C05467=1086.034,-74.611,447.064,174.286,17.662,152.886
C05468=1086.028,-74.861,447.075,174.284,17.661,152.887
C05469=1086.021,-75.111,447.086,174.282,17.660,152.887
C05470=1086.016,-75.360,447.097,174.281,17.658,152.887
C05471=1086.010,-75.610,447.108,174.279,17.657,152.887
C05472=1086.004,-75.860,447.119,174.278,17.656,152.887
C05473=1085.998,-76.110,447.130,174.277,17.655,152.887
C05474=1085.992,-76.359,447.141,174.275,17.654,152.887
C05475=1085.986,-76.608,447.151,174.274,17.653,152.887
C05476=1085.979,-76.858,447.162,174.272,17.652,152.887
C05477=1085.974,-77.108,447.173,174.271,17.650,152.887
C05478=1085.968,-77.358,447.183,174.269,17.649,152.887
C05479=1085.962,-77.607,447.194,174.268,17.648,152.887
C05480=1085.956,-77.858,447.205,174.266,17.646,152.887
C05481=1085.950,-78.107,447.215,174.265,17.645,152.887
C05482=1085.944,-78.356,447.226,174.263,17.644,152.887
C05483=1085.938,-78.607,447.238,174.261,17.643,152.887
C05484=1085.932,-78.856,447.248,174.260,17.642,152.887
C05485=1085.926,-79.105,447.259,174.258,17.640,152.887
C05486=1085.921,-79.356,447.270,174.257,17.639,152.887
C05487=1085.914,-79.605,447.280,174.255,17.638,152.888
C05488=1085.908,-79.855,447.291,174.254,17.636,152.888
C05489=1085.902,-80.104,447.302,174.252,17.635,152.888
C05490=1085.896,-80.354,447.313,174.250,17.634,152.888
C05491=1085.889,-80.604,447.323,174.250,17.634,152.888
C05492=1085.883,-80.879,447.335,174.247,17.631,152.888
C05493=1085.876,-81.154,447.346,174.246,17.630,152.888
C05494=1085.870,-81.429,447.358,174.244,17.629,152.888
C05495=1085.863,-81.705,447.371,174.243,17.628,152.888
C05496=1085.857,-81.955,447.381,174.241,17.627,152.888
C05497=1085.851,-82.204,447.391,174.239,17.626,152.888
C05498=1085.845,-82.454,447.402,174.238,17.625,152.888
C05499=1085.839,-82.704,447.413,174.236,17.623,152.888
C05500=1085.832,-82.953,447.423,174.235,17.622,152.888
C05501=1085.827,-83.203,447.434,174.233,17.621,152.889
C05502=1085.820,-83.452,447.444,174.232,17.620,152.889
C05503=1085.814,-83.703,447.455,174.231,17.619,152.889
C05504=1085.808,-83.952,447.466,174.229,17.618,152.889
C05505=1085.802,-84.202,447.476,174.227,17.617,152.889
C05506=1085.796,-84.451,447.486,174.226,17.616,152.889
C05507=1085.790,-84.702,447.498,174.224,17.615,152.889
C05508=1085.784,-84.951,447.507,174.223,17.613,152.889
C05509=1085.778,-85.201,447.518,174.221,17.612,152.889
C05510=1085.771,-85.450,447.528,174.219,17.611,152.889
C05511=1085.766,-85.699,447.539,174.218,17.610,152.889
C05512=1085.760,-85.950,447.550,174.216,17.608,152.889
C05513=1085.753,-86.199,447.560,174.216,17.608,152.889
C05514=1085.747,-86.449,447.571,174.214,17.607,152.889
C05515=1085.741,-86.699,447.581,174.212,17.606,152.890
C05516=1085.736,-86.948,447.591,174.211,17.604,152.890
C05517=1085.729,-87.198,447.603,174.209,17.603,152.890
C05518=1085.723,-87.448,447.612,174.208,17.602,152.890
C05519=1085.717,-87.698,447.623,174.206,17.601,152.890
C05520=1085.711,-87.947,447.633,174.204,17.600,152.890
C05521=1085.705,-88.197,447.644,174.203,17.599,152.890
C05522=1085.699,-88.446,447.654,174.201,17.597,152.890
C05523=1085.693,-88.697,447.664,174.200,17.596,152.890
C05524=1085.687,-88.947,447.675,174.199,17.595,152.890
C05525=1085.681,-89.196,447.686,174.197,17.594,152.890
C05526=1085.675,-89.446,447.696,174.195,17.593,152.890
C05527=1085.669,-89.695,447.706,174.194,17.592,152.891
C05528=1085.663,-89.945,447.716,174.192,17.591,152.891
C05529=1085.656,-90.195,447.727,174.191,17.590,152.891
C05530=1085.650,-90.444,447.738,174.189,17.589,152.891
C05531=1085.645,-90.695,447.748,174.187,17.587,152.891
C05532=1085.639,-90.944,447.758,174.187,17.587,152.891
C05533=1085.633,-91.194,447.768,174.185,17.586,152.891
C05534=1085.627,-91.443,447.779,174.183,17.585,152.891
C05535=1085.621,-91.693,447.789,174.182,17.583,152.891
C05536=1085.615,-91.942,447.799,174.180,17.582,152.891
C05537=1085.609,-92.193,447.810,174.179,17.581,152.891
C05538=1085.602,-92.442,447.820,174.177,17.580,152.891
C05539=1085.597,-92.692,447.830,174.175,17.579,152.892
C05540=1085.590,-92.942,447.840,174.174,17.578,152.892
C05541=1085.585,-93.192,447.850,174.173,17.577,152.892
C05542=1085.578,-93.441,447.861,174.171,17.576,152.892
C05543=1085.573,-93.691,447.871,174.170,17.575,152.892
C05544=1085.567,-93.940,447.881,174.168,17.574,152.892
C05545=1085.561,-94.190,447.891,174.166,17.573,152.892
C05546=1085.555,-94.439,447.902,174.165,17.572,152.892
C05547=1085.549,-94.690,447.912,174.163,17.570,152.892
C05548=1085.543,-94.939,447.922,174.162,17.570,152.892
C05549=1085.537,-95.189,447.932,174.161,17.569,152.892
C05550=1085.530,-95.439,447.943,174.159,17.568,152.893
C05551=1085.525,-95.689,447.953,174.157,17.567,152.893
C05552=1085.518,-95.938,447.963,174.156,17.566,152.893
C05553=1085.513,-96.188,447.973,174.154,17.564,152.893
C05554=1085.507,-96.438,447.983,174.153,17.563,152.893
C05555=1085.501,-96.687,447.994,174.152,17.563,152.893
C05556=1085.494,-96.964,448.005,174.150,17.561,152.893
C05557=1085.488,-97.242,448.016,174.148,17.560,152.893
C05558=1085.481,-97.520,448.028,174.146,17.559,152.893
C05559=1085.474,-97.797,448.038,174.144,17.558,152.893
C05560=1085.469,-98.047,448.049,174.144,17.557,152.894
C05561=1085.462,-98.297,448.059,174.142,17.556,152.894
C05562=1085.455,-98.547,448.069,174.140,17.555,152.894
C05563=1085.450,-98.797,448.079,174.139,17.554,152.894
C05564=1085.444,-99.046,448.089,174.137,17.553,152.894
C05565=1085.437,-99.296,448.099,174.135,17.552,152.894
C05566=1085.432,-99.546,448.109,174.134,17.551,152.894
C05567=1085.425,-99.795,448.119,174.133,17.550,152.894
C05568=1085.419,-100.045,448.129,174.131,17.549,152.894
C05569=1085.414,-100.295,448.139,174.129,17.548,152.894
C05570=1085.407,-100.544,448.149,174.128,17.547,152.895
C05571=1085.401,-100.794,448.159,174.126,17.546,152.895
C05572=1085.395,-101.044,448.168,174.125,17.546,152.895
C05573=1085.389,-101.293,448.179,174.123,17.545,152.895
C05574=1085.383,-101.543,448.189,174.122,17.544,152.895
C05575=1085.377,-101.793,448.198,174.120,17.543,152.895
C05576=1085.371,-102.043,448.208,174.118,17.542,152.895
C05577=1085.365,-102.292,448.219,174.117,17.541,152.895
C05578=1085.359,-102.542,448.228,174.116,17.540,152.896
C05579=1085.353,-102.792,448.238,174.114,17.539,152.896
C05580=1085.347,-103.041,448.249,174.113,17.538,152.896
C05581=1085.341,-103.291,448.258,174.111,17.537,152.896
C05582=1085.335,-103.541,448.268,174.109,17.536,152.896
C05583=1085.328,-103.791,448.278,174.108,17.535,152.896
C05584=1085.323,-104.041,448.288,174.107,17.535,152.896
C05585=1085.317,-104.290,448.298,174.105,17.534,152.896
C05586=1085.310,-104.540,448.308,174.103,17.533,152.897
C05587=1085.304,-104.789,448.317,174.102,17.532,152.897
C05588=1085.298,-105.039,448.327,174.100,17.531,152.897
C05589=1085.292,-105.289,448.338,174.099,17.530,152.897
C05590=1085.286,-105.538,448.347,174.097,17.529,152.897
C05591=1085.280,-105.788,448.357,174.096,17.528,152.897
C05592=1085.274,-106.038,448.366,174.094,17.527,152.897
C05593=1085.268,-106.288,448.376,174.092,17.526,152.897
C05594=1085.262,-106.537,448.387,174.091,17.526,152.898
C05595=1085.256,-106.787,448.396,174.090,17.525,152.898
C05596=1085.250,-107.037,448.406,174.088,17.524,152.898
C05597=1085.243,-107.287,448.415,174.086,17.523,152.898
C05598=1085.237,-107.537,448.425,174.084,17.522,152.898
C05599=1085.232,-107.787,448.435,174.084,17.522,152.898
C05600=1085.226,-108.036,448.445,174.082,17.521,152.898
C05601=1085.219,-108.286,448.455,174.080,17.519,152.898
C05602=1085.213,-108.535,448.465,174.079,17.518,152.899
C05603=1085.207,-108.785,448.474,174.078,17.518,152.899
C05604=1085.201,-109.035,448.484,174.076,17.517,152.899
C05605=1085.194,-109.285,448.493,174.074,17.516,152.899
C05606=1085.188,-109.535,448.503,174.073,17.515,152.899
C05607=1085.182,-109.784,448.512,174.071,17.515,152.899
C05608=1085.176,-110.034,448.522,174.070,17.514,152.899
C05609=1085.169,-110.283,448.532,174.068,17.513,152.900
C05610=1085.164,-110.534,448.542,174.067,17.512,152.900
C05611=1085.158,-110.783,448.552,174.065,17.511,152.900
C05612=1085.152,-111.033,448.562,174.064,17.511,152.900
C05613=1085.145,-111.283,448.571,174.062,17.510,152.900
C05614=1085.139,-111.533,448.581,174.060,17.509,152.900
C05615=1085.133,-111.783,448.590,174.059,17.508,152.900
C05616=1085.128,-112.032,448.600,174.057,17.507,152.901
C05617=1085.121,-112.281,448.609,174.056,17.507,152.901
C05618=1085.115,-112.531,448.619,174.054,17.506,152.901
C05619=1085.109,-112.781,448.628,174.052,17.505,152.901
C05620=1085.103,-113.054,448.639,174.051,17.504,152.901
C05621=1085.095,-113.327,448.650,174.049,17.503,152.901
C05622=1085.089,-113.600,448.660,174.047,17.502,152.902
C05623=1085.082,-113.873,448.670,174.046,17.501,152.902
C05624=1085.076,-114.123,448.680,174.045,17.501,152.902
C05625=1085.070,-114.373,448.689,174.043,17.500,152.902
C05626=1085.064,-114.622,448.699,174.041,17.499,152.902
C05627=1085.058,-114.872,448.708,174.040,17.498,152.902
C05628=1085.052,-115.122,448.718,174.038,17.498,152.902
C05629=1085.046,-115.371,448.727,174.037,17.497,152.903
C05630=1085.040,-115.621,448.737,174.035,17.497,152.903
C05631=1085.033,-115.871,448.746,174.033,17.495,152.903
C05632=1085.027,-116.121,448.756,174.032,17.495,152.903
C05633=1085.021,-116.371,448.766,174.030,17.494,152.903
C05634=1085.015,-116.620,448.775,174.029,17.493,152.903
C05635=1085.009,-116.870,448.785,174.027,17.492,152.903
C05636=1085.003,-117.120,448.793,174.026,17.492,152.904
C05637=1084.997,-117.370,448.803,174.024,17.491,152.904
C05638=1084.990,-117.619,448.812,174.022,17.491,152.904
C05639=1084.984,-117.869,448.821,174.022,17.490,152.904
C05640=1084.978,-118.119,448.831,174.020,17.489,152.904
C05641=1084.972,-118.369,448.840,174.018,17.489,152.905
C05642=1084.966,-118.618,448.850,174.016,17.487,152.905
C05643=1084.959,-118.868,448.860,174.015,17.487,152.905
C05644=1084.954,-119.117,448.869,174.014,17.486,152.905
C05645=1084.948,-119.367,448.878,174.012,17.486,152.905
C05646=1084.942,-119.617,448.887,174.010,17.485,152.905
C05647=1084.936,-119.867,448.897,174.009,17.484,152.905
C05648=1084.929,-120.117,448.906,174.007,17.484,152.906
C05649=1084.923,-120.367,448.915,174.006,17.483,152.906
C05650=1084.916,-120.616,448.925,174.004,17.483,152.906
C05651=1084.911,-120.865,448.934,174.003,17.482,152.906
C05652=1084.905,-121.116,448.943,174.001,17.481,152.906
C05653=1084.899,-121.366,448.952,173.999,17.480,152.906
C05654=1084.893,-121.615,448.962,173.998,17.480,152.907
C05655=1084.886,-121.865,448.971,173.996,17.479,152.907
C05656=1084.880,-122.115,448.981,173.995,17.478,152.907
C05657=1084.874,-122.364,448.990,173.994,17.478,152.907
C05658=1084.868,-122.614,448.999,173.992,17.477,152.907
C05659=1084.862,-122.864,449.008,173.990,17.476,152.908
C05660=1084.856,-123.114,449.018,173.988,17.476,152.908
C05661=1084.849,-123.363,449.027,173.987,17.475,152.908
C05662=1084.843,-123.614,449.036,173.985,17.475,152.908
C05663=1084.837,-123.863,449.045,173.984,17.474,152.908
C05664=1084.831,-124.113,449.054,173.983,17.474,152.908
C05665=1084.825,-124.362,449.064,173.981,17.472,152.909
C05666=1084.819,-124.613,449.073,173.979,17.472,152.909
C05667=1084.812,-124.862,449.082,173.978,17.471,152.909
C05668=1084.807,-125.111,449.091,173.976,17.471,152.909
C05669=1084.801,-125.361,449.101,173.975,17.470,152.909
C05670=1084.794,-125.611,449.109,173.973,17.469,152.910
C05671=1084.788,-125.861,449.118,173.972,17.469,152.910
C05672=1084.782,-126.111,449.128,173.970,17.468,152.910
C05673=1084.775,-126.361,449.137,173.968,17.468,152.910
C05674=1084.769,-126.610,449.145,173.967,17.467,152.910
C05675=1084.763,-126.860,449.155,173.965,17.467,152.910
C05676=1084.757,-127.110,449.165,173.963,17.466,152.911
C05677=1084.750,-127.360,449.173,173.963,17.466,152.911
C05678=1084.744,-127.610,449.182,173.961,17.465,152.911
C05679=1084.739,-127.859,449.192,173.959,17.464,152.911
C05680=1084.733,-128.116,449.201,173.958,17.464,152.911
C05681=1084.731,-128.373,449.211,173.957,17.462,152.911
C05682=1084.733,-128.628,449.224,173.956,17.459,152.911
C05683=1084.740,-128.881,449.237,173.955,17.454,152.910
C05684=1084.338,-128.903,449.105,173.912,17.569,152.940
C05685=1084.332,-128.650,449.091,173.912,17.573,152.941
C05686=1084.328,-128.394,449.079,173.912,17.577,152.941
C05687=1084.331,-128.138,449.068,173.914,17.578,152.941
C05688=1084.335,-127.881,449.059,173.915,17.579,152.941
C05689=1084.342,-127.632,449.050,173.917,17.580,152.941
C05690=1084.348,-127.382,449.040,173.918,17.580,152.941
C05691=1084.354,-127.132,449.031,173.920,17.581,152.941
C05692=1084.361,-126.882,449.022,173.922,17.582,152.941
C05693=1084.367,-126.633,449.013,173.923,17.582,152.940
C05694=1084.373,-126.383,449.004,173.925,17.583,152.940
C05695=1084.379,-126.133,448.995,173.927,17.584,152.940
C05696=1084.386,-125.883,448.986,173.928,17.584,152.940
C05697=1084.392,-125.633,448.977,173.929,17.585,152.940
C05698=1084.397,-125.384,448.968,173.931,17.585,152.939
C05699=1084.404,-125.134,448.959,173.933,17.586,152.939
C05700=1084.410,-124.884,448.949,173.934,17.586,152.939
C05701=1084.416,-124.634,448.940,173.936,17.587,152.939
C05702=1084.422,-124.384,448.931,173.938,17.588,152.939
C05703=1084.428,-124.135,448.922,173.938,17.588,152.939
C05704=1084.435,-123.886,448.913,173.940,17.589,152.938
C05705=1084.441,-123.635,448.904,173.942,17.590,152.938
C05706=1084.447,-123.385,448.894,173.944,17.590,152.938
C05707=1084.453,-123.136,448.885,173.945,17.591,152.938
C05708=1084.459,-122.886,448.875,173.947,17.592,152.938
C05709=1084.466,-122.637,448.867,173.948,17.593,152.937
C05710=1084.471,-122.387,448.858,173.949,17.593,152.937
C05711=1084.478,-122.137,448.848,173.951,17.594,152.937
C05712=1084.484,-121.887,448.839,173.953,17.594,152.937
C05713=1084.490,-121.637,448.829,173.955,17.595,152.937
C05714=1084.496,-121.387,448.819,173.956,17.595,152.937
C05715=1084.501,-121.138,448.811,173.957,17.596,152.936
C05716=1084.508,-120.888,448.802,173.959,17.597,152.936
C05717=1084.514,-120.638,448.792,173.961,17.598,152.936
C05718=1084.521,-120.389,448.783,173.962,17.598,152.936
C05719=1084.527,-120.139,448.773,173.964,17.599,152.936
C05720=1084.533,-119.889,448.764,173.965,17.600,152.936
C05721=1084.538,-119.639,448.755,173.966,17.601,152.936
C05722=1084.544,-119.390,448.746,173.968,17.601,152.935
C05723=1084.551,-119.140,448.736,173.970,17.602,152.935
C05724=1084.557,-118.890,448.727,173.972,17.603,152.935
C05725=1084.564,-118.640,448.718,173.973,17.603,152.935
C05726=1084.570,-118.391,448.708,173.975,17.604,152.935
C05727=1084.576,-118.141,448.698,173.976,17.605,152.934
C05728=1084.582,-117.891,448.689,173.978,17.606,152.934
C05729=1084.588,-117.642,448.680,173.979,17.606,152.934
C05730=1084.594,-117.392,448.671,173.981,17.607,152.934
C05731=1084.600,-117.142,448.661,173.982,17.608,152.934
C05732=1084.606,-116.892,448.652,173.984,17.608,152.934
C05733=1084.612,-116.642,448.642,173.985,17.609,152.934
C05734=1084.618,-116.392,448.632,173.987,17.610,152.933
C05735=1084.624,-116.143,448.623,173.989,17.611,152.933
C05736=1084.631,-115.893,448.613,173.990,17.612,152.933
C05737=1084.638,-115.643,448.604,173.991,17.612,152.933
C05738=1084.643,-115.394,448.595,173.993,17.613,152.933
C05739=1084.649,-115.144,448.586,173.995,17.614,152.933
C05740=1084.655,-114.895,448.576,173.996,17.615,152.932
C05741=1084.662,-114.645,448.566,173.998,17.615,152.932
C05742=1084.668,-114.395,448.557,173.999,17.616,152.932
C05743=1084.674,-114.145,448.547,174.001,17.617,152.932
C05744=1084.680,-113.895,448.538,174.003,17.617,152.932
C05745=1084.686,-113.622,448.527,174.004,17.619,152.932
C05746=1084.693,-113.348,448.516,174.005,17.619,152.932
C05747=1084.700,-113.075,448.506,174.007,17.620,152.931
C05748=1084.706,-112.802,448.496,174.009,17.621,152.931
C05749=1084.712,-112.552,448.486,174.011,17.622,152.931
C05750=1084.718,-112.303,448.477,174.012,17.623,152.931
C05751=1084.725,-112.053,448.467,174.014,17.624,152.931
C05752=1084.731,-111.803,448.458,174.015,17.624,152.931
C05753=1084.737,-111.553,448.448,174.017,17.625,152.931
C05754=1084.743,-111.303,448.438,174.018,17.626,152.930
C05755=1084.749,-111.054,448.429,174.020,17.627,152.930
C05756=1084.755,-110.804,448.419,174.022,17.628,152.930
C05757=1084.762,-110.555,448.409,174.023,17.628,152.930
C05758=1084.768,-110.305,448.399,174.024,17.629,152.930
C05759=1084.774,-110.055,448.390,174.026,17.630,152.930
C05760=1084.780,-109.805,448.380,174.028,17.631,152.929
C05761=1084.786,-109.555,448.370,174.029,17.631,152.929
C05762=1084.791,-109.306,448.361,174.030,17.632,152.929
C05763=1084.798,-109.056,448.351,174.032,17.633,152.929
C05764=1084.804,-108.806,448.342,174.034,17.634,152.929
C05765=1084.810,-108.557,448.332,174.036,17.635,152.929
C05766=1084.816,-108.307,448.322,174.036,17.635,152.929
C05767=1084.823,-108.058,448.312,174.038,17.637,152.929
C05768=1084.829,-107.808,448.303,174.040,17.638,152.929
C05769=1084.835,-107.558,448.293,174.041,17.639,152.928
C05770=1084.840,-107.308,448.283,174.043,17.640,152.928
C05771=1084.846,-107.058,448.274,174.044,17.640,152.928
C05772=1084.853,-106.808,448.264,174.046,17.641,152.928
C05773=1084.859,-106.559,448.254,174.048,17.642,152.928
C05774=1084.865,-106.309,448.244,174.049,17.643,152.928
C05775=1084.871,-106.060,448.235,174.051,17.644,152.928
C05776=1084.877,-105.809,448.224,174.052,17.644,152.928
C05777=1084.883,-105.560,448.215,174.053,17.646,152.927
C05778=1084.890,-105.311,448.205,174.055,17.647,152.927
C05779=1084.896,-105.061,448.195,174.057,17.648,152.927
C05780=1084.901,-104.811,448.185,174.059,17.648,152.927
C05781=1084.907,-104.561,448.175,174.059,17.649,152.927
C05782=1084.913,-104.311,448.166,174.061,17.650,152.927
C05783=1084.920,-104.062,448.155,174.063,17.651,152.927
C05784=1084.925,-103.812,448.145,174.064,17.652,152.927
C05785=1084.932,-103.562,448.136,174.066,17.653,152.926
C05786=1084.938,-103.312,448.126,174.068,17.654,152.926
C05787=1084.944,-103.063,448.116,174.069,17.654,152.926
C05788=1084.950,-102.813,448.106,174.070,17.656,152.926
C05789=1084.956,-102.563,448.096,174.072,17.657,152.926
C05790=1084.962,-102.313,448.087,174.074,17.658,152.926
C05791=1084.968,-102.064,448.076,174.075,17.659,152.926
C05792=1084.974,-101.814,448.066,174.076,17.659,152.926
C05793=1084.980,-101.564,448.056,174.078,17.660,152.926
C05794=1084.987,-101.315,448.046,174.079,17.661,152.926
C05795=1084.993,-101.065,448.037,174.081,17.662,152.925
C05796=1084.998,-100.815,448.026,174.083,17.663,152.925
C05797=1085.005,-100.566,448.016,174.084,17.665,152.925
C05798=1085.011,-100.316,448.007,174.085,17.665,152.925
C05799=1085.016,-100.066,447.996,174.087,17.666,152.925
C05800=1085.023,-99.816,447.986,174.088,17.667,152.925
C05801=1085.030,-99.566,447.976,174.090,17.668,152.925
C05802=1085.036,-99.316,447.967,174.092,17.669,152.925
C05803=1085.041,-99.067,447.956,174.093,17.670,152.925
C05804=1085.048,-98.817,447.946,174.095,17.671,152.924
C05805=1085.054,-98.567,447.937,174.096,17.672,152.924
C05806=1085.059,-98.318,447.926,174.098,17.673,152.924
C05807=1085.066,-98.068,447.916,174.099,17.674,152.924
C05808=1085.072,-97.818,447.907,174.101,17.675,152.924
C05809=1085.078,-97.540,447.895,174.103,17.676,152.924
C05810=1085.085,-97.263,447.884,174.104,17.677,152.924
C05811=1085.091,-96.986,447.872,174.106,17.678,152.924
C05812=1085.098,-96.708,447.861,174.108,17.679,152.924
C05813=1085.104,-96.458,447.851,174.109,17.680,152.923
C05814=1085.110,-96.209,447.841,174.111,17.681,152.923
C05815=1085.116,-95.959,447.831,174.113,17.682,152.923
C05816=1085.122,-95.709,447.820,174.114,17.684,152.923
C05817=1085.128,-95.459,447.810,174.115,17.685,152.923
C05818=1085.134,-95.210,447.800,174.116,17.686,152.923
C05819=1085.140,-94.959,447.789,174.118,17.687,152.923
C05820=1085.146,-94.709,447.780,174.120,17.688,152.923
C05821=1085.152,-94.460,447.769,174.121,17.689,152.923
C05822=1085.158,-94.210,447.759,174.123,17.690,152.923
C05823=1085.164,-93.961,447.748,174.124,17.691,152.923
C05824=1085.170,-93.711,447.739,174.126,17.693,152.923
C05825=1085.176,-93.461,447.728,174.127,17.693,152.922
C05826=1085.182,-93.212,447.718,174.129,17.694,152.922
C05827=1085.188,-92.962,447.708,174.130,17.695,152.922
C05828=1085.194,-92.712,447.698,174.132,17.696,152.922
C05829=1085.200,-92.463,447.687,174.134,17.697,152.922
C05830=1085.206,-92.213,447.677,174.135,17.699,152.922
C05831=1085.212,-91.963,447.666,174.137,17.700,152.922
C05832=1085.218,-91.713,447.657,174.138,17.701,152.922
C05833=1085.224,-91.464,447.646,174.139,17.701,152.922
C05834=1085.231,-91.214,447.636,174.141,17.703,152.922
C05835=1085.236,-90.964,447.625,174.142,17.704,152.922
C05836=1085.243,-90.715,447.615,174.144,17.705,152.922
C05837=1085.248,-90.465,447.605,174.145,17.706,152.921
C05838=1085.254,-90.215,447.594,174.147,17.707,152.921
C05839=1085.261,-89.965,447.584,174.149,17.708,152.921
C05840=1085.266,-89.715,447.573,174.150,17.710,152.921
C05841=1085.273,-89.466,447.563,174.152,17.711,152.921
C05842=1085.278,-89.216,447.553,174.153,17.712,152.921
C05843=1085.285,-88.967,447.542,174.154,17.713,152.921
C05844=1085.290,-88.717,447.532,174.156,17.714,152.921
C05845=1085.296,-88.467,447.521,174.157,17.715,152.921
C05846=1085.303,-88.218,447.511,174.159,17.716,152.921
C05847=1085.308,-87.967,447.501,174.161,17.717,152.921
C05848=1085.315,-87.718,447.490,174.162,17.718,152.921
C05849=1085.321,-87.469,447.479,174.164,17.720,152.921
C05850=1085.327,-87.219,447.470,174.165,17.721,152.921
C05851=1085.333,-86.969,447.459,174.167,17.722,152.920
C05852=1085.339,-86.719,447.448,174.168,17.723,152.920
C05853=1085.345,-86.469,447.438,174.170,17.724,152.920
C05854=1085.351,-86.220,447.427,174.171,17.725,152.920
C05855=1085.357,-85.971,447.417,174.173,17.726,152.920
C05856=1085.363,-85.720,447.407,174.174,17.727,152.920
C05857=1085.369,-85.470,447.396,174.176,17.729,152.920
C05858=1085.375,-85.221,447.385,174.177,17.730,152.920
C05859=1085.381,-84.971,447.375,174.179,17.731,152.920
C05860=1085.387,-84.722,447.365,174.181,17.732,152.920
C05861=1085.394,-84.472,447.354,174.182,17.734,152.920
C05862=1085.399,-84.222,447.343,174.184,17.735,152.920
C05863=1085.406,-83.973,447.333,174.185,17.736,152.920
C05864=1085.411,-83.723,447.322,174.186,17.736,152.919
C05865=1085.418,-83.473,447.311,174.188,17.738,152.920
C05866=1085.424,-83.224,447.301,174.189,17.739,152.919
C05867=1085.430,-82.974,447.291,174.191,17.740,152.919
C05868=1085.436,-82.724,447.280,174.192,17.742,152.919
C05869=1085.442,-82.474,447.269,174.194,17.743,152.919
C05870=1085.448,-82.225,447.258,174.196,17.744,152.919
C05871=1085.454,-81.975,447.249,174.197,17.745,152.919
C05872=1085.460,-81.725,447.238,174.199,17.746,152.919
C05873=1085.467,-81.450,447.226,174.200,17.747,152.919
C05874=1085.474,-81.175,447.214,174.202,17.748,152.919
C05875=1085.480,-80.899,447.203,174.203,17.750,152.919
C05876=1085.487,-80.624,447.190,174.205,17.751,152.919
C05877=1085.493,-80.374,447.179,174.207,17.752,152.919
C05878=1085.500,-80.125,447.169,174.208,17.754,152.919
C05879=1085.506,-79.874,447.159,174.210,17.755,152.919
C05880=1085.511,-79.625,447.148,174.211,17.756,152.918
C05881=1085.517,-79.375,447.137,174.213,17.757,152.918
C05882=1085.524,-79.126,447.127,174.214,17.758,152.918
C05883=1085.530,-78.876,447.115,174.216,17.760,152.918
C05884=1085.536,-78.626,447.104,174.218,17.761,152.918
C05885=1085.541,-78.377,447.094,174.219,17.762,152.918
C05886=1085.547,-78.127,447.083,174.221,17.764,152.918
C05887=1085.553,-77.876,447.072,174.222,17.765,152.918
C05888=1085.560,-77.627,447.062,174.224,17.766,152.918
C05889=1085.565,-77.378,447.051,174.225,17.767,152.918
C05890=1085.572,-77.128,447.040,174.227,17.769,152.918
C05891=1085.577,-76.878,447.029,174.228,17.770,152.918
C05892=1085.583,-76.629,447.018,174.230,17.771,152.918
C05893=1085.589,-76.379,447.007,174.231,17.773,152.918
C05894=1085.596,-76.129,446.997,174.232,17.773,152.918
C05895=1085.602,-75.880,446.986,174.234,17.775,152.918
C05896=1085.608,-75.630,446.975,174.235,17.776,152.918
C05897=1085.614,-75.380,446.964,174.237,17.777,152.918
C05898=1085.620,-75.131,446.953,174.238,17.778,152.918
C05899=1085.625,-74.881,446.942,174.240,17.780,152.918
C05900=1085.631,-74.632,446.931,174.241,17.781,152.918
C05901=1085.637,-74.381,446.920,174.243,17.782,152.917
C05902=1085.644,-74.132,446.909,174.244,17.784,152.918
C05903=1085.649,-73.882,446.899,174.246,17.785,152.917
C05904=1085.656,-73.632,446.888,174.247,17.786,152.917
C05905=1085.661,-73.382,446.876,174.249,17.788,152.918
C05906=1085.666,-73.133,446.866,174.251,17.789,152.917
C05907=1085.672,-72.884,446.854,174.252,17.791,152.917
C05908=1085.679,-72.634,446.843,174.254,17.792,152.917
C05909=1085.685,-72.384,446.832,174.255,17.793,152.917
C05910=1085.690,-72.135,446.821,174.257,17.794,152.917
C05911=1085.697,-71.884,446.810,174.258,17.796,152.917
C05912=1085.702,-71.635,446.799,174.259,17.797,152.917
C05913=1085.708,-71.385,446.788,174.261,17.798,152.917
C05914=1085.714,-71.136,446.777,174.262,17.800,152.917
C05915=1085.720,-70.886,446.766,174.264,17.801,152.917
C05916=1085.726,-70.636,446.755,174.266,17.803,152.917
C05917=1085.732,-70.387,446.744,174.267,17.804,152.917
C05918=1085.738,-70.137,446.733,174.269,17.805,152.917
C05919=1085.744,-69.887,446.722,174.270,17.807,152.917
C05920=1085.749,-69.637,446.711,174.272,17.808,152.917
C05921=1085.755,-69.387,446.699,174.273,17.809,152.917
C05922=1085.761,-69.138,446.688,174.275,17.811,152.917
C05923=1085.767,-68.889,446.677,174.276,17.812,152.917
C05924=1085.773,-68.639,446.666,174.277,17.814,152.917
C05925=1085.779,-68.389,446.655,174.279,17.815,152.917
C05926=1085.785,-68.140,446.644,174.281,17.816,152.917
C05927=1085.791,-67.889,446.633,174.282,17.817,152.917
C05928=1085.797,-67.640,446.622,174.284,17.819,152.917
C05929=1085.802,-67.390,446.610,174.285,17.821,152.917
C05930=1085.808,-67.141,446.598,174.287,17.822,152.917
C05931=1085.814,-66.891,446.587,174.288,17.823,152.917
C05932=1085.820,-66.642,446.577,174.290,17.824,152.917
C05933=1085.826,-66.391,446.565,174.291,17.826,152.917
C05934=1085.832,-66.142,446.554,174.292,17.827,152.917
C05935=1085.839,-65.892,446.542,174.294,17.828,152.917
C05936=1085.844,-65.643,446.532,174.296,17.830,152.917
C05937=1085.851,-65.369,446.519,174.297,17.832,152.917
C05938=1085.857,-65.096,446.506,174.299,17.833,152.917
C05939=1085.864,-64.823,446.494,174.301,17.835,152.917
C05940=1085.869,-64.550,446.482,174.302,17.836,152.917
C05941=1085.876,-64.300,446.470,174.304,17.837,152.917
C05942=1085.882,-64.051,446.459,174.305,17.839,152.917
C05943=1085.888,-63.800,446.448,174.307,17.840,152.917
C05944=1085.894,-63.551,446.437,174.308,17.842,152.917
C05945=1085.900,-63.302,446.426,174.310,17.843,152.917
C05946=1085.905,-63.052,446.414,174.311,17.845,152.917
C05947=1085.911,-62.802,446.403,174.313,17.846,152.917
C05948=1085.917,-62.552,446.392,174.314,17.847,152.917
C05949=1085.924,-62.303,446.380,174.316,17.849,152.917
C05950=1085.930,-62.053,446.369,174.317,17.850,152.917
C05951=1085.935,-61.803,446.358,174.319,17.852,152.917
C05952=1085.941,-61.553,446.346,174.320,17.853,152.916
C05953=1085.947,-61.304,446.335,174.322,17.854,152.916
C05954=1085.953,-61.055,446.324,174.323,17.856,152.917
C05955=1085.960,-60.805,446.312,174.325,17.857,152.916
C05956=1085.965,-60.555,446.300,174.326,17.858,152.916
C05957=1085.971,-60.305,446.289,174.328,17.860,152.916
C05958=1085.977,-60.056,446.278,174.329,17.861,152.916
C05959=1085.983,-59.806,446.266,174.331,17.863,152.916
C05960=1085.989,-59.557,446.255,174.333,17.865,152.916
C05961=1085.995,-59.307,446.243,174.334,17.866,152.916
C05962=1086.001,-59.057,446.232,174.336,17.867,152.916
C05963=1086.007,-58.807,446.220,174.337,17.869,152.916
C05964=1086.013,-58.558,446.209,174.339,17.870,152.916
C05965=1086.020,-58.308,446.197,174.340,17.871,152.916
C05966=1086.025,-58.059,446.186,174.342,17.873,152.916
C05967=1086.031,-57.808,446.174,174.343,17.875,152.916
C05968=1086.037,-57.560,446.163,174.345,17.876,152.916
C05969=1086.043,-57.309,446.152,174.346,17.877,152.916
C05970=1086.049,-57.060,446.139,174.348,17.879,152.916
C05971=1086.055,-56.810,446.128,174.349,17.880,152.916
C05972=1086.061,-56.561,446.117,174.351,17.881,152.916
C05973=1086.068,-56.311,446.105,174.352,17.883,152.916
C05974=1086.073,-56.061,446.093,174.354,17.884,152.916
C05975=1086.079,-55.812,446.082,174.355,17.886,152.916
C05976=1086.086,-55.561,446.071,174.356,17.887,152.916
C05977=1086.092,-55.312,446.059,174.358,17.889,152.916
C05978=1086.097,-55.062,446.047,174.360,17.890,152.916
C05979=1086.103,-54.813,446.036,174.361,17.891,152.916
C05980=1086.110,-54.564,446.024,174.362,17.893,152.916
C05981=1086.115,-54.313,446.012,174.365,17.895,152.916
C05982=1086.121,-54.064,446.000,174.366,17.896,152.916
C05983=1086.128,-53.814,445.989,174.368,17.898,152.916
C05984=1086.134,-53.565,445.977,174.369,17.899,152.916
C05985=1086.139,-53.315,445.966,174.371,17.900,152.916
C05986=1086.146,-53.066,445.954,174.372,17.902,152.916
C05987=1086.152,-52.816,445.943,174.373,17.903,152.916
C05988=1086.158,-52.566,445.930,174.375,17.905,152.916
C05989=1086.164,-52.316,445.919,174.377,17.906,152.916
C05990=1086.170,-52.067,445.907,174.378,17.908,152.916
C05991=1086.176,-51.818,445.896,174.379,17.909,152.916
C05992=1086.182,-51.567,445.884,174.381,17.910,152.916
C05993=1086.188,-51.318,445.872,174.382,17.912,152.916
C05994=1086.194,-51.068,445.861,174.384,17.913,152.916
C05995=1086.200,-50.818,445.849,174.385,17.915,152.916
C05996=1086.207,-50.569,445.837,174.388,17.917,152.916
C05997=1086.212,-50.319,445.826,174.389,17.918,152.916
C05998=1086.218,-50.069,445.813,174.390,17.920,152.916
C05999=1086.224,-49.820,445.801,174.392,17.921,152.916
C06000=1086.230,-49.570,445.790,174.394,17.922,152.916
C06001=1086.236,-49.298,445.776,174.395,17.924,152.916
C06002=1086.242,-49.026,445.764,174.396,17.926,152.916
C06003=1086.249,-48.754,445.751,174.399,17.928,152.916
C06004=1086.256,-48.483,445.738,174.400,17.929,152.916
C06005=1086.261,-48.233,445.726,174.401,17.931,152.916
C06006=1086.267,-47.984,445.714,174.403,17.932,152.916
C06007=1086.273,-47.734,445.702,174.404,17.934,152.916
C06008=1086.279,-47.483,445.690,174.406,17.935,152.916
C06009=1086.285,-47.234,445.678,174.407,17.937,152.916
C06010=1086.291,-46.985,445.666,174.409,17.939,152.916
C06011=1086.297,-46.736,445.654,174.411,17.940,152.916
C06012=1086.303,-46.485,445.642,174.412,17.942,152.916
C06013=1086.308,-46.235,445.630,174.414,17.943,152.916
C06014=1086.314,-45.986,445.618,174.415,17.945,152.916
C06015=1086.320,-45.736,445.607,174.416,17.946,152.916
C06016=1086.326,-45.487,445.595,174.418,17.948,152.917
C06017=1086.332,-45.237,445.582,174.419,17.950,152.917
C06018=1086.339,-44.988,445.570,174.421,17.951,152.916
C06019=1086.344,-44.738,445.558,174.422,17.952,152.916
C06020=1086.350,-44.488,445.546,174.424,17.954,152.916
C06021=1086.356,-44.238,445.534,174.426,17.956,152.917
C06022=1086.362,-43.989,445.522,174.427,17.957,152.917
C06023=1086.367,-43.739,445.510,174.429,17.959,152.917
C06024=1086.374,-43.490,445.498,174.430,17.961,152.917
C06025=1086.379,-43.240,445.486,174.431,17.962,152.917
C06026=1086.386,-42.990,445.474,174.433,17.963,152.917
C06027=1086.392,-42.740,445.462,174.435,17.965,152.917
C06028=1086.397,-42.491,445.450,174.436,17.966,152.917
C06029=1086.404,-42.242,445.438,174.438,17.968,152.917
C06030=1086.410,-41.992,445.425,174.440,17.970,152.917
C06031=1086.415,-41.742,445.414,174.441,17.972,152.917
C06032=1086.421,-41.492,445.402,174.442,17.973,152.917
C06033=1086.427,-41.243,445.389,174.444,17.975,152.917
C06034=1086.432,-40.993,445.377,174.445,17.976,152.917
C06035=1086.439,-40.744,445.365,174.447,17.977,152.917
C06036=1086.445,-40.494,445.352,174.448,17.979,152.917
C06037=1086.452,-40.244,445.340,174.450,17.981,152.917
C06038=1086.457,-39.995,445.328,174.452,17.983,152.917
C06039=1086.463,-39.745,445.316,174.453,17.984,152.917
C06040=1086.469,-39.496,445.304,174.455,17.986,152.917
C06041=1086.474,-39.246,445.292,174.456,17.987,152.917
C06042=1086.480,-38.996,445.280,174.457,17.989,152.917
C06043=1086.487,-38.746,445.268,174.459,17.990,152.917
C06044=1086.493,-38.497,445.255,174.460,17.992,152.917
C06045=1086.498,-38.247,445.243,174.463,17.994,152.917
C06046=1086.504,-37.997,445.230,174.464,17.995,152.917
C06047=1086.510,-37.748,445.218,174.466,17.997,152.917
C06048=1086.515,-37.498,445.206,174.467,17.998,152.917
C06049=1086.522,-37.249,445.194,174.468,18.000,152.917
C06050=1086.528,-36.999,445.181,174.470,18.001,152.917
C06051=1086.533,-36.750,445.169,174.471,18.003,152.917
C06052=1086.539,-36.500,445.156,174.473,18.005,152.917
C06053=1086.545,-36.250,445.144,174.475,18.007,152.917
C06054=1086.551,-36.000,445.131,174.476,18.008,152.917
C06055=1086.557,-35.751,445.120,174.478,18.010,152.917
C06056=1086.563,-35.501,445.107,174.479,18.011,152.917
C06057=1086.569,-35.251,445.095,174.480,18.013,152.917
C06058=1086.574,-35.002,445.082,174.482,18.015,152.917
C06059=1086.580,-34.752,445.070,174.484,18.017,152.917
C06060=1086.586,-34.503,445.057,174.485,18.018,152.917
C06061=1086.592,-34.253,445.045,174.487,18.020,152.917
C06062=1086.597,-34.004,445.032,174.488,18.021,152.918
C06063=1086.604,-33.755,445.020,174.490,18.023,152.918
C06064=1086.610,-33.505,445.007,174.491,18.024,152.918
C06065=1086.616,-33.233,444.994,174.493,18.027,152.918
C06066=1086.623,-32.961,444.981,174.495,18.028,152.918
C06067=1086.629,-32.690,444.966,174.496,18.030,152.918
C06068=1086.635,-32.418,444.953,174.498,18.032,152.918
C06069=1086.641,-32.169,444.940,174.500,18.033,152.918
C06070=1086.647,-31.919,444.928,174.501,18.035,152.918
C06071=1086.653,-31.669,444.916,174.502,18.036,152.918
C06072=1086.659,-31.420,444.904,174.504,18.038,152.918
C06073=1086.665,-31.171,444.890,174.505,18.040,152.918
C06074=1086.671,-30.921,444.878,174.507,18.042,152.918
C06075=1086.677,-30.671,444.865,174.509,18.043,152.918
C06076=1086.683,-30.421,444.853,174.510,18.045,152.918
C06077=1086.688,-30.172,444.840,174.512,18.046,152.918
C06078=1086.694,-29.922,444.828,174.513,18.048,152.918
C06079=1086.700,-29.673,444.815,174.514,18.050,152.918
C06080=1086.706,-29.423,444.802,174.517,18.052,152.918
C06081=1086.712,-29.173,444.790,174.518,18.053,152.918
C06082=1086.718,-28.923,444.778,174.519,18.055,152.918
C06083=1086.724,-28.675,444.765,174.521,18.056,152.918
C06084=1086.730,-28.425,444.752,174.522,18.058,152.918
C06085=1086.736,-28.175,444.740,174.524,18.059,152.918
C06086=1086.742,-27.925,444.727,174.526,18.062,152.918
C06087=1086.748,-27.676,444.714,174.527,18.063,152.918
C06088=1086.754,-27.426,444.701,174.529,18.065,152.918
C06089=1086.760,-27.176,444.689,174.530,18.066,152.918
C06090=1086.766,-26.926,444.676,174.532,18.068,152.918
C06091=1086.771,-26.678,444.663,174.533,18.069,152.918
C06092=1086.777,-26.428,444.651,174.535,18.071,152.918
C06093=1086.783,-26.178,444.638,174.537,18.073,152.919
C06094=1086.789,-25.928,444.624,174.538,18.075,152.919
C06095=1086.795,-25.678,444.612,174.539,18.077,152.919
C06096=1086.800,-25.429,444.599,174.541,18.078,152.919
C06097=1086.806,-25.179,444.587,174.542,18.080,152.919
C06098=1086.812,-24.930,444.574,174.544,18.082,152.919
C06099=1086.818,-24.680,444.561,174.546,18.083,152.919
C06100=1086.824,-24.430,444.549,174.547,18.085,152.919
C06101=1086.830,-24.181,444.535,174.548,18.087,152.919
C06102=1086.835,-23.931,444.522,174.550,18.088,152.919
C06103=1086.841,-23.682,444.509,174.552,18.090,152.919
C06104=1086.847,-23.432,444.497,174.553,18.092,152.919
C06105=1086.853,-23.182,444.484,174.555,18.093,152.919
C06106=1086.859,-22.933,444.471,174.556,18.095,152.919
C06107=1086.865,-22.683,444.458,174.558,18.097,152.919
C06108=1086.870,-22.434,444.444,174.560,18.099,152.919
C06109=1086.876,-22.184,444.432,174.561,18.101,152.919
C06110=1086.882,-21.934,444.419,174.562,18.102,152.919
C06111=1086.888,-21.685,444.406,174.564,18.104,152.919
C06112=1086.894,-21.436,444.394,174.565,18.105,152.919
C06113=1086.900,-21.186,444.381,174.567,18.107,152.920
C06114=1086.905,-20.936,444.367,174.569,18.109,152.920
C06115=1086.911,-20.687,444.354,174.570,18.111,152.920
C06116=1086.917,-20.437,444.342,174.572,18.112,152.920
C06117=1086.923,-20.187,444.329,174.573,18.114,152.920
C06118=1086.929,-19.938,444.316,174.574,18.115,152.920
C06119=1086.934,-19.688,444.303,174.577,18.117,152.920
C06120=1086.941,-19.438,444.289,174.578,18.119,152.920
C06121=1086.946,-19.188,444.277,174.579,18.121,152.920
C06122=1086.953,-18.939,444.264,174.581,18.123,152.920
C06123=1086.959,-18.689,444.251,174.582,18.124,152.920
C06124=1086.964,-18.440,444.237,174.584,18.126,152.920
C06125=1086.970,-18.191,444.224,174.586,18.128,152.920
C06126=1086.976,-17.941,444.212,174.587,18.129,152.920
C06127=1086.982,-17.692,444.198,174.588,18.131,152.920
C06128=1086.988,-17.442,444.186,174.591,18.133,152.920
C06129=1086.994,-17.169,444.172,174.592,18.135,152.920
C06130=1087.000,-16.897,444.157,174.593,18.136,152.920
C06131=1087.007,-16.625,444.142,174.596,18.138,152.920
C06132=1087.013,-16.352,444.129,174.597,18.140,152.920
C06133=1087.019,-16.103,444.115,174.598,18.142,152.920
C06134=1087.025,-15.854,444.102,174.601,18.144,152.920
C06135=1087.031,-15.604,444.089,174.602,18.146,152.920
C06136=1087.037,-15.354,444.076,174.603,18.147,152.921
C06137=1087.042,-15.104,444.063,174.605,18.149,152.921
C06138=1087.049,-14.855,444.049,174.606,18.150,152.921
C06139=1087.055,-14.606,444.036,174.608,18.152,152.921
C06140=1087.060,-14.356,444.023,174.610,18.154,152.921
C06141=1087.066,-14.106,444.010,174.611,18.155,152.921
C06142=1087.072,-13.857,443.996,174.612,18.158,152.921
C06143=1087.078,-13.607,443.983,174.615,18.160,152.921
C06144=1087.083,-13.357,443.969,174.616,18.161,152.921
C06145=1087.089,-13.108,443.956,174.617,18.163,152.921
C06146=1087.095,-12.858,443.944,174.619,18.164,152.921
C06147=1087.101,-12.608,443.930,174.620,18.166,152.921
C06148=1087.107,-12.359,443.916,174.622,18.168,152.921
C06149=1087.112,-12.109,443.903,174.624,18.170,152.921
C06150=1087.118,-11.860,443.890,174.625,18.172,152.921
C06151=1087.124,-11.610,443.876,174.626,18.173,152.921
C06152=1087.130,-11.360,443.864,174.629,18.175,152.921
C06153=1087.136,-11.111,443.850,174.630,18.177,152.921
C06154=1087.141,-10.861,443.836,174.631,18.178,152.921
C06155=1087.148,-10.612,443.823,174.633,18.180,152.921
C06156=1087.153,-10.362,443.810,174.635,18.182,152.921
C06157=1087.159,-10.113,443.797,174.636,18.184,152.922
C06158=1087.164,-9.863,443.783,174.638,18.186,152.922
C06159=1087.171,-9.614,443.770,174.639,18.187,152.922
C06160=1087.176,-9.364,443.756,174.640,18.189,152.922
C06161=1087.182,-9.114,443.743,174.643,18.191,152.922
C06162=1087.188,-8.865,443.729,174.644,18.192,152.922
C06163=1087.194,-8.616,443.716,174.645,18.194,152.922
C06164=1087.199,-8.366,443.702,174.647,18.196,152.922
C06165=1087.206,-8.116,443.689,174.649,18.198,152.922
C06166=1087.212,-7.866,443.676,174.650,18.199,152.922
C06167=1087.217,-7.617,443.662,174.652,18.201,152.922
C06168=1087.224,-7.367,443.649,174.653,18.203,152.922
C06169=1087.229,-7.118,443.635,174.655,18.205,152.922
C06170=1087.235,-6.869,443.622,174.657,18.207,152.922
C06171=1087.241,-6.619,443.608,174.658,18.208,152.922
C06172=1087.247,-6.370,443.595,174.659,18.210,152.922
C06173=1087.252,-6.119,443.582,174.662,18.212,152.922
C06174=1087.258,-5.870,443.568,174.663,18.213,152.922
C06175=1087.264,-5.621,443.554,174.665,18.215,152.922
C06176=1087.270,-5.370,443.540,174.666,18.217,152.923
C06177=1087.276,-5.121,443.527,174.668,18.219,152.923
C06178=1087.282,-4.872,443.513,174.669,18.221,152.923
C06179=1087.288,-4.622,443.500,174.671,18.222,152.923
C06180=1087.293,-4.373,443.486,174.672,18.224,152.923
C06181=1087.300,-4.123,443.473,174.674,18.226,152.923
C06182=1087.305,-3.874,443.459,174.676,18.227,152.923
C06183=1087.312,-3.624,443.445,174.677,18.229,152.923
C06184=1087.317,-3.374,443.431,174.679,18.230,152.923
C06185=1087.324,-3.125,443.418,174.681,18.233,152.923
C06186=1087.329,-2.875,443.404,174.682,18.235,152.923
C06187=1087.334,-2.626,443.390,174.683,18.236,152.923
C06188=1087.340,-2.376,443.376,174.685,18.238,152.923
C06189=1087.346,-2.127,443.363,174.687,18.240,152.923
C06190=1087.352,-1.877,443.349,174.688,18.241,152.923
C06191=1087.357,-1.628,443.335,174.690,18.243,152.923
C06192=1087.363,-1.378,443.322,174.691,18.245,152.923
C06193=1087.369,-1.103,443.307,174.693,18.247,152.923
C06194=1087.376,-0.830,443.292,174.695,18.249,152.923
C06195=1087.382,-0.556,443.277,174.697,18.251,152.924
C06196=1087.388,-0.282,443.261,174.698,18.253,152.924
C06197=1087.394,-0.032,443.247,174.700,18.255,152.924
C06198=1087.399,0.217,443.234,174.702,18.256,152.924
C06199=1087.405,0.467,443.220,174.703,18.258,152.924
C06200=1087.411,0.716,443.206,174.704,18.260,152.924
C06201=1087.417,0.966,443.192,174.706,18.262,152.924
C06202=1087.423,1.216,443.178,174.708,18.264,152.924
C06203=1087.428,1.466,443.164,174.709,18.265,152.924
C06204=1087.434,1.715,443.150,174.712,18.267,152.924
C06205=1087.440,1.964,443.137,174.713,18.269,152.924
C06206=1087.446,2.213,443.123,174.714,18.271,152.924
C06207=1087.451,2.463,443.109,174.716,18.273,152.924
C06208=1087.457,2.713,443.095,174.718,18.275,152.924
C06209=1087.463,2.963,443.081,174.719,18.276,152.924
C06210=1087.469,3.212,443.067,174.721,18.278,152.924
C06211=1087.475,3.461,443.053,174.722,18.279,152.924
C06212=1087.480,3.711,443.039,174.724,18.282,152.925
C06213=1087.486,3.961,443.025,174.725,18.283,152.925
C06214=1087.492,4.210,443.011,174.727,18.285,152.925
C06215=1087.497,4.460,442.997,174.729,18.287,152.925
C06216=1087.504,4.709,442.983,174.730,18.289,152.925
C06217=1087.509,4.958,442.969,174.732,18.290,152.925
C06218=1087.515,5.209,442.955,174.733,18.292,152.925
C06219=1087.521,5.458,442.941,174.735,18.294,152.925
C06220=1087.526,5.708,442.927,174.737,18.296,152.925
C06221=1087.532,5.957,442.913,174.738,18.298,152.925
C06222=1087.539,6.207,442.899,174.740,18.300,152.925
C06223=1087.544,6.456,442.885,174.742,18.301,152.925
C06224=1087.550,6.706,442.871,174.743,18.303,152.925
C06225=1087.555,6.955,442.857,174.744,18.304,152.925
C06226=1087.561,7.205,442.843,174.747,18.306,152.925
C06227=1087.567,7.455,442.829,174.748,18.308,152.925
C06228=1087.573,7.704,442.814,174.749,18.310,152.925
C06229=1087.578,7.953,442.800,174.752,18.312,152.925
C06230=1087.585,8.203,442.787,174.753,18.314,152.925
C06231=1087.591,8.452,442.772,174.754,18.315,152.926
C06232=1087.596,8.702,442.758,174.756,18.317,152.926
C06233=1087.602,8.951,442.744,174.758,18.319,152.926
C06234=1087.608,9.201,442.729,174.759,18.320,152.926
C06235=1087.614,9.450,442.715,174.761,18.322,152.926
C06236=1087.619,9.700,442.702,174.763,18.325,152.926
C06237=1087.625,9.950,442.687,174.764,18.326,152.926
C06238=1087.631,10.199,442.673,174.766,18.328,152.926
C06239=1087.637,10.448,442.660,174.768,18.330,152.926
C06240=1087.644,10.698,442.645,174.769,18.331,152.926
C06241=1087.649,10.948,442.631,174.771,18.333,152.926
C06242=1087.655,11.197,442.616,174.772,18.334,152.926
C06243=1087.661,11.447,442.602,174.774,18.336,152.926
C06244=1087.666,11.697,442.588,174.776,18.338,152.926
C06245=1087.672,11.945,442.573,174.777,18.340,152.926
C06246=1087.678,12.196,442.559,174.779,18.342,152.926
C06247=1087.684,12.445,442.545,174.781,18.344,152.926
C06248=1087.689,12.694,442.531,174.782,18.345,152.926
C06249=1087.696,12.944,442.516,174.784,18.347,152.926
C06250=1087.701,13.194,442.502,174.786,18.349,152.926
C06251=1087.707,13.442,442.487,174.787,18.351,152.926
C06252=1087.713,13.693,442.473,174.788,18.352,152.927
C06253=1087.719,13.942,442.459,174.791,18.354,152.927
C06254=1087.725,14.192,442.444,174.792,18.356,152.927
C06255=1087.731,14.441,442.430,174.794,18.357,152.927
C06256=1087.736,14.691,442.416,174.796,18.359,152.927
C06257=1087.743,14.967,442.400,174.797,18.361,152.927
C06258=1087.750,15.243,442.383,174.799,18.363,152.927
C06259=1087.757,15.518,442.368,174.801,18.365,152.927
C06260=1087.763,15.795,442.352,174.803,18.367,152.927
C06261=1087.767,16.044,442.338,174.804,18.369,152.927
C06262=1087.773,16.293,442.323,174.806,18.371,152.927
C06263=1087.780,16.543,442.308,174.808,18.373,152.927
C06264=1087.785,16.793,442.294,174.809,18.374,152.927
C06265=1087.792,17.042,442.279,174.811,18.376,152.927
C06266=1087.797,17.292,442.265,174.813,18.378,152.927
C06267=1087.803,17.541,442.251,174.814,18.380,152.927
C06268=1087.808,17.791,442.235,174.816,18.381,152.927
C06269=1087.814,18.040,442.221,174.818,18.383,152.927
C06270=1087.820,18.289,442.207,174.819,18.385,152.927
C06271=1087.826,18.540,442.193,174.821,18.386,152.927
C06272=1087.832,18.789,442.178,174.823,18.389,152.928
C06273=1087.838,19.038,442.163,174.824,18.390,152.928
C06274=1087.843,19.288,442.149,174.825,18.392,152.928
C06275=1087.848,19.537,442.134,174.828,18.394,152.928
C06276=1087.855,19.787,442.119,174.829,18.396,152.928
C06277=1087.860,20.036,442.105,174.830,18.397,152.928
C06278=1087.867,20.286,442.090,174.833,18.399,152.928
C06279=1087.872,20.535,442.076,174.834,18.401,152.928
C06280=1087.878,20.785,442.061,174.836,18.402,152.928
C06281=1087.884,21.034,442.046,174.838,18.404,152.928
C06282=1087.889,21.283,442.032,174.839,18.407,152.928
C06283=1087.895,21.533,442.016,174.840,18.408,152.928
C06284=1087.900,21.783,442.002,174.843,18.410,152.928
C06285=1087.907,22.033,441.987,174.844,18.412,152.928
C06286=1087.913,22.282,441.973,174.845,18.413,152.928
C06287=1087.918,22.531,441.958,174.848,18.415,152.928
C06288=1087.924,22.781,441.943,174.849,18.417,152.928
C06289=1087.930,23.030,441.929,174.850,18.418,152.928
C06290=1087.935,23.280,441.913,174.853,18.421,152.928
C06291=1087.941,23.529,441.899,174.854,18.422,152.928
C06292=1087.947,23.779,441.885,174.856,18.424,152.928
C06293=1087.952,24.028,441.869,174.858,18.426,152.928
C06294=1087.958,24.278,441.854,174.859,18.428,152.929
C06295=1087.964,24.527,441.840,174.861,18.430,152.929
C06296=1087.971,24.777,441.825,174.863,18.431,152.929
C06297=1087.976,25.026,441.810,174.864,18.433,152.929
C06298=1087.982,25.276,441.795,174.866,18.435,152.929
C06299=1087.988,25.525,441.781,174.868,18.437,152.929
C06300=1087.993,25.775,441.765,174.869,18.438,152.929
C06301=1087.999,26.024,441.751,174.871,18.440,152.929
C06302=1088.005,26.274,441.736,174.873,18.442,152.929
C06303=1088.010,26.523,441.721,174.874,18.443,152.929
C06304=1088.017,26.773,441.706,174.876,18.445,152.929
C06305=1088.022,27.023,441.691,174.878,18.447,152.929
C06306=1088.028,27.272,441.676,174.879,18.449,152.929
C06307=1088.034,27.521,441.662,174.882,18.451,152.929
C06308=1088.039,27.771,441.646,174.883,18.452,152.929
C06309=1088.045,28.020,441.632,174.884,18.454,152.929
C06310=1088.051,28.270,441.617,174.886,18.456,152.929
C06311=1088.057,28.519,441.601,174.888,18.458,152.929
C06312=1088.063,28.769,441.587,174.889,18.459,152.929
C06313=1088.068,29.018,441.571,174.891,18.461,152.929
C06314=1088.074,29.268,441.556,174.893,18.463,152.929
C06315=1088.079,29.517,441.541,174.895,18.465,152.929
C06316=1088.086,29.767,441.526,174.896,18.467,152.929
C06317=1088.091,30.016,441.511,174.898,18.468,152.929
C06318=1088.097,30.266,441.496,174.900,18.470,152.929
C06319=1088.102,30.515,441.481,174.902,18.472,152.929
C06320=1088.109,30.764,441.466,174.903,18.473,152.930
C06321=1088.115,31.042,441.449,174.905,18.475,152.930
C06322=1088.121,31.319,441.432,174.907,18.478,152.930
C06323=1088.127,31.596,441.415,174.909,18.480,152.930
C06324=1088.133,31.874,441.399,174.911,18.482,152.930
C06325=1088.140,32.123,441.384,174.912,18.483,152.930
C06326=1088.145,32.373,441.368,174.915,18.485,152.930
C06327=1088.151,32.622,441.353,174.916,18.487,152.930
C06328=1088.157,32.872,441.338,174.917,18.488,152.930
C06329=1088.162,33.121,441.323,174.920,18.491,152.930
C06330=1088.168,33.371,441.308,174.921,18.492,152.930
C06331=1088.173,33.620,441.293,174.923,18.494,152.930
C06332=1088.180,33.870,441.278,174.925,18.496,152.930
C06333=1088.185,34.120,441.262,174.926,18.497,152.930
C06334=1088.191,34.369,441.248,174.928,18.499,152.930
C06335=1088.197,34.618,441.231,174.930,18.501,152.930
C06336=1088.202,34.867,441.216,174.931,18.502,152.930
C06337=1088.209,35.117,441.201,174.933,18.504,152.930
C06338=1088.214,35.367,441.186,174.935,18.506,152.930
C06339=1088.220,35.616,441.171,174.937,18.508,152.930
C06340=1088.226,35.866,441.156,174.939,18.510,152.930
C06341=1088.232,36.114,441.140,174.940,18.511,152.930
C06342=1088.237,36.364,441.125,174.942,18.513,152.930
C06343=1088.243,36.614,441.109,174.944,18.515,152.930
C06344=1088.249,36.863,441.095,174.945,18.516,152.930
C06345=1088.254,37.113,441.079,174.947,18.518,152.930
C06346=1088.261,37.362,441.063,174.949,18.520,152.930
C06347=1088.266,37.612,441.048,174.951,18.522,152.930
C06348=1088.272,37.861,441.033,174.952,18.524,152.930
C06349=1088.278,38.111,441.018,174.954,18.525,152.931
C06350=1088.284,38.360,441.002,174.956,18.527,152.931
C06351=1088.289,38.610,440.986,174.957,18.529,152.931
C06352=1088.294,38.859,440.971,174.960,18.531,152.931
C06353=1088.301,39.109,440.956,174.961,18.532,152.931
C06354=1088.307,39.358,440.940,174.963,18.534,152.931
C06355=1088.312,39.607,440.925,174.965,18.536,152.931
C06356=1088.317,39.857,440.909,174.966,18.538,152.931
C06357=1088.324,40.106,440.894,174.968,18.540,152.931
C06358=1088.329,40.356,440.878,174.970,18.541,152.931
C06359=1088.335,40.606,440.863,174.971,18.543,152.931
C06360=1088.341,40.855,440.847,174.974,18.545,152.931
C06361=1088.346,41.104,440.831,174.975,18.546,152.931
C06362=1088.352,41.354,440.816,174.977,18.548,152.931
C06363=1088.358,41.603,440.800,174.979,18.550,152.931
C06364=1088.363,41.852,440.785,174.980,18.552,152.931
C06365=1088.369,42.102,440.769,174.982,18.554,152.931
C06366=1088.375,42.352,440.753,174.984,18.555,152.931
C06367=1088.380,42.601,440.739,174.986,18.557,152.931
C06368=1088.386,42.851,440.723,174.987,18.559,152.931
C06369=1088.392,43.100,440.707,174.989,18.560,152.931
C06370=1088.397,43.349,440.692,174.991,18.562,152.931
C06371=1088.403,43.599,440.675,174.993,18.564,152.931
C06372=1088.409,43.848,440.660,174.995,18.566,152.931
C06373=1088.415,44.098,440.644,174.996,18.567,152.931
C06374=1088.420,44.347,440.629,174.998,18.569,152.931
C06375=1088.426,44.597,440.613,175.000,18.571,152.931
C06376=1088.431,44.846,440.598,175.001,18.572,152.931
C06377=1088.437,45.095,440.582,175.004,18.574,152.931
C06378=1088.443,45.345,440.566,175.005,18.576,152.931
C06379=1088.449,45.595,440.550,175.007,18.578,152.931
C06380=1088.454,45.843,440.534,175.009,18.580,152.931
C06381=1088.460,46.093,440.519,175.010,18.581,152.931
C06382=1088.466,46.343,440.503,175.013,18.583,152.931
C06383=1088.471,46.592,440.487,175.014,18.585,152.931
C06384=1088.477,46.841,440.471,175.016,18.587,152.931
C06385=1088.482,47.119,440.453,175.018,18.588,152.932
C06386=1088.489,47.396,440.436,175.020,18.590,152.932
C06387=1088.495,47.674,440.418,175.022,18.593,152.932
C06388=1088.502,47.951,440.400,175.023,18.595,152.932
C06389=1088.507,48.201,440.385,175.026,18.597,152.932
C06390=1088.513,48.450,440.369,175.027,18.598,152.932
C06391=1088.518,48.700,440.353,175.029,18.600,152.932
C06392=1088.524,48.949,440.337,175.031,18.601,152.932
C06393=1088.530,49.198,440.321,175.033,18.603,152.932
C06394=1088.535,49.448,440.306,175.035,18.605,152.932
C06395=1088.541,49.697,440.289,175.036,18.606,152.932
C06396=1088.547,49.947,440.274,175.038,18.609,152.932
C06397=1088.552,50.196,440.258,175.040,18.610,152.932
C06398=1088.558,50.445,440.242,175.042,18.612,152.932
C06399=1088.564,50.695,440.226,175.043,18.614,152.932
C06400=1088.570,50.944,440.210,175.046,18.616,152.932
C06401=1088.575,51.194,440.193,175.047,18.617,152.932
C06402=1088.580,51.443,440.178,175.049,18.619,152.932
C06403=1088.586,51.693,440.162,175.051,18.620,152.932
C06404=1088.592,51.942,440.145,175.052,18.622,152.932
C06405=1088.598,52.192,440.130,175.055,18.624,152.932
C06406=1088.603,52.441,440.114,175.056,18.626,152.932
C06407=1088.609,52.690,440.098,175.058,18.628,152.932
C06408=1088.615,52.939,440.081,175.060,18.629,152.932
C06409=1088.620,53.189,440.066,175.062,18.631,152.932
C06410=1088.626,53.439,440.050,175.064,18.632,152.932
C06411=1088.632,53.688,440.033,175.065,18.634,152.932
C06412=1088.638,53.937,440.017,175.067,18.636,152.932
C06413=1088.643,54.187,440.001,175.069,18.637,152.932
C06414=1088.649,54.436,439.985,175.071,18.640,152.932
C06415=1088.654,54.686,439.969,175.072,18.641,152.932
C06416=1088.660,54.935,439.953,175.075,18.643,152.932
C06417=1088.666,55.184,439.936,175.076,18.644,152.932
C06418=1088.672,55.434,439.921,175.079,18.646,152.932
C06419=1088.678,55.684,439.904,175.080,18.648,152.932
C06420=1088.683,55.932,439.889,175.082,18.650,152.932
C06421=1088.689,56.182,439.872,175.084,18.651,152.932
C06422=1088.695,56.431,439.855,175.085,18.652,152.932
C06423=1088.700,56.681,439.839,175.088,18.655,152.932
C06424=1088.706,56.931,439.824,175.089,18.656,152.932
C06425=1088.712,57.180,439.807,175.091,18.658,152.932
C06426=1088.718,57.429,439.791,175.093,18.659,152.932
C06427=1088.724,57.679,439.775,175.095,18.661,152.932
C06428=1088.729,57.928,439.758,175.097,18.663,152.932
C06429=1088.735,58.178,439.742,175.099,18.665,152.932
C06430=1088.741,58.427,439.726,175.101,18.666,152.932
C06431=1088.747,58.676,439.709,175.102,18.667,152.932
C06432=1088.752,58.925,439.693,175.104,18.670,152.932
C06433=1088.758,59.174,439.677,175.106,18.671,152.932
C06434=1088.764,59.424,439.660,175.108,18.673,152.932
C06435=1088.769,59.673,439.644,175.110,18.674,152.932
C06436=1088.775,59.923,439.629,175.112,18.676,152.932
C06437=1088.781,60.173,439.612,175.114,18.677,152.932
C06438=1088.787,60.422,439.596,175.116,18.679,152.932
C06439=1088.792,60.672,439.579,175.117,18.681,152.932
C06440=1088.798,60.921,439.563,175.119,18.683,152.932
C06441=1088.804,61.170,439.547,175.121,18.684,152.932
C06442=1088.810,61.420,439.530,175.123,18.686,152.932
C06443=1088.816,61.669,439.514,175.125,18.688,152.932
C06444=1088.822,61.918,439.497,175.126,18.689,152.932
C06445=1088.828,62.167,439.480,175.129,18.691,152.932
C06446=1088.833,62.417,439.464,175.130,18.692,152.932
C06447=1088.839,62.666,439.448,175.133,18.694,152.932
C06448=1088.845,62.916,439.431,175.134,18.695,152.932
C06449=1088.852,63.193,439.413,175.136,18.697,152.932
C06450=1088.858,63.471,439.395,175.139,18.699,152.932
C06451=1088.865,63.748,439.377,175.141,18.701,152.932
C06452=1088.871,64.025,439.358,175.143,18.703,152.932
C06453=1088.877,64.275,439.342,175.145,18.704,152.932
C06454=1088.882,64.524,439.324,175.146,18.706,152.932
C06455=1088.888,64.773,439.308,175.149,18.708,152.932
C06456=1088.894,65.022,439.292,175.150,18.709,152.932
C06457=1088.900,65.272,439.275,175.153,18.711,152.932
C06458=1088.906,65.521,439.259,175.154,18.712,152.932
C06459=1088.911,65.771,439.242,175.156,18.715,152.932
C06460=1088.917,66.020,439.226,175.158,18.716,152.932
C06461=1088.922,66.269,439.208,175.160,18.718,152.932
C06462=1088.928,66.519,439.192,175.162,18.719,152.932
C06463=1088.934,66.768,439.176,175.164,18.721,152.931
C06464=1088.939,67.018,439.159,175.166,18.722,152.932
C06465=1088.945,67.267,439.143,175.168,18.724,152.932
C06466=1088.951,67.516,439.125,175.170,18.725,152.931
C06467=1088.957,67.765,439.109,175.172,18.727,152.931
C06468=1088.962,68.015,439.092,175.173,18.729,152.932
C06469=1088.968,68.264,439.076,175.176,18.731,152.931
C06470=1088.973,68.513,439.058,175.177,18.732,152.931
C06471=1088.979,68.763,439.042,175.179,18.734,152.931
C06472=1088.985,69.012,439.025,175.181,18.735,152.931
C06473=1088.991,69.262,439.009,175.183,18.737,152.931
C06474=1088.996,69.511,438.991,175.185,18.738,152.931
C06475=1089.002,69.760,438.975,175.187,18.740,152.931
C06476=1089.007,70.010,438.958,175.189,18.742,152.931
C06477=1089.014,70.259,438.941,175.191,18.744,152.931
C06478=1089.019,70.509,438.924,175.193,18.745,152.931
C06479=1089.025,70.758,438.908,175.195,18.747,152.931
C06480=1089.031,71.007,438.890,175.197,18.748,152.931
C06481=1089.036,71.257,438.873,175.199,18.750,152.931
C06482=1089.042,71.506,438.857,175.200,18.752,152.931
C06483=1089.047,71.755,438.839,175.203,18.753,152.931
C06484=1089.053,72.005,438.823,175.204,18.755,152.931
C06485=1089.059,72.254,438.806,175.207,18.756,152.931
C06486=1089.064,72.503,438.789,175.208,18.758,152.931
C06487=1089.070,72.753,438.772,175.210,18.760,152.931
C06488=1089.076,73.002,438.755,175.212,18.761,152.931
C06489=1089.081,73.251,438.738,175.214,18.763,152.931
C06490=1089.087,73.502,438.721,175.216,18.764,152.931
C06491=1089.093,73.751,438.704,175.218,18.766,152.931
C06492=1089.099,74.000,438.688,175.220,18.768,152.931
C06493=1089.104,74.249,438.670,175.222,18.769,152.931
C06494=1089.110,74.499,438.653,175.224,18.771,152.931
C06495=1089.116,74.747,438.636,175.226,18.772,152.931
C06496=1089.121,74.997,438.619,175.228,18.774,152.931
C06497=1089.127,75.246,438.602,175.230,18.776,152.931
C06498=1089.133,75.496,438.585,175.232,18.777,152.931
C06499=1089.139,75.745,438.568,175.234,18.779,152.931
C06500=1089.144,75.995,438.551,175.235,18.780,152.931
C06501=1089.149,76.244,438.533,175.238,18.782,152.931
C06502=1089.155,76.493,438.517,175.239,18.783,152.931
C06503=1089.161,76.742,438.499,175.242,18.785,152.931
C06504=1089.166,76.992,438.482,175.243,18.786,152.930
C06505=1089.173,77.241,438.465,175.246,18.789,152.930
C06506=1089.178,77.491,438.448,175.247,18.790,152.930
C06507=1089.184,77.740,438.431,175.250,18.792,152.930
C06508=1089.190,77.989,438.414,175.251,18.793,152.930
C06509=1089.195,78.238,438.397,175.253,18.795,152.930
C06510=1089.201,78.488,438.379,175.255,18.796,152.930
C06511=1089.206,78.738,438.362,175.257,18.798,152.930
C06512=1089.212,78.987,438.345,175.260,18.799,152.930
C06513=1089.218,79.264,438.325,175.261,18.801,152.930
C06514=1089.225,79.541,438.307,175.264,18.803,152.930
C06515=1089.230,79.818,438.287,175.266,18.805,152.930
C06516=1089.237,80.095,438.268,175.268,18.807,152.930
C06517=1089.243,80.344,438.250,175.270,18.808,152.930
C06518=1089.248,80.594,438.233,175.272,18.810,152.930
C06519=1089.254,80.844,438.216,175.274,18.811,152.930
C06520=1089.260,81.092,438.199,175.276,18.813,152.930
C06521=1089.265,81.342,438.182,175.278,18.814,152.930
C06522=1089.271,81.591,438.164,175.280,18.816,152.930
C06523=1089.276,81.840,438.147,175.283,18.818,152.930
C06524=1089.282,82.091,438.129,175.284,18.819,152.930
C06525=1089.288,82.340,438.112,175.287,18.821,152.930
C06526=1089.293,82.589,438.094,175.288,18.822,152.930
C06527=1089.299,82.838,438.077,175.291,18.824,152.929
C06528=1089.304,83.087,438.060,175.292,18.825,152.930
C06529=1089.310,83.337,438.042,175.295,18.827,152.929
C06530=1089.316,83.586,438.024,175.296,18.828,152.929
C06531=1089.322,83.835,438.007,175.298,18.830,152.929
C06532=1089.327,84.084,437.991,175.300,18.831,152.929
C06533=1089.333,84.334,437.973,175.302,18.833,152.929
C06534=1089.339,84.583,437.955,175.305,18.835,152.929
C06535=1089.344,84.832,437.937,175.306,18.836,152.929
C06536=1089.350,85.081,437.920,175.309,18.838,152.929
C06537=1089.356,85.332,437.903,175.311,18.839,152.929
C06538=1089.361,85.581,437.885,175.313,18.841,152.929
C06539=1089.367,85.830,437.868,175.314,18.842,152.929
C06540=1089.373,86.080,437.850,175.317,18.844,152.929
C06541=1089.378,86.329,437.832,175.318,18.845,152.929
C06542=1089.384,86.578,437.814,175.321,18.846,152.929
C06543=1089.389,86.827,437.797,175.322,18.848,152.929
C06544=1089.395,87.076,437.779,175.325,18.850,152.929
C06545=1089.401,87.326,437.762,175.327,18.851,152.928
C06546=1089.406,87.575,437.745,175.329,18.853,152.928
C06547=1089.412,87.825,437.727,175.331,18.854,152.928
C06548=1089.418,88.074,437.709,175.333,18.855,152.928
C06549=1089.423,88.323,437.691,175.335,18.857,152.928
C06550=1089.429,88.573,437.674,175.337,18.858,152.928
C06551=1089.435,88.822,437.656,175.339,18.860,152.928
C06552=1089.440,89.071,437.638,175.342,18.862,152.928
C06553=1089.447,89.320,437.620,175.343,18.863,152.928
C06554=1089.452,89.570,437.603,175.346,18.865,152.928
C06555=1089.458,89.819,437.585,175.347,18.866,152.928
C06556=1089.464,90.068,437.567,175.350,18.868,152.928
C06557=1089.469,90.317,437.550,175.352,18.869,152.928
C06558=1089.475,90.567,437.532,175.354,18.870,152.928
C06559=1089.481,90.816,437.514,175.355,18.872,152.928
C06560=1089.486,91.065,437.497,175.358,18.873,152.927
C06561=1089.492,91.315,437.479,175.361,18.875,152.927
C06562=1089.497,91.564,437.461,175.362,18.877,152.927
C06563=1089.503,91.813,437.443,175.364,18.878,152.927
C06564=1089.509,92.063,437.425,175.366,18.879,152.927
C06565=1089.514,92.312,437.408,175.368,18.881,152.927
C06566=1089.520,92.561,437.390,175.371,18.883,152.927
C06567=1089.526,92.811,437.371,175.373,18.884,152.927
C06568=1089.531,93.060,437.353,175.375,18.886,152.927
C06569=1089.537,93.309,437.336,175.377,18.887,152.927
C06570=1089.543,93.558,437.318,175.379,18.888,152.927
C06571=1089.548,93.808,437.300,175.380,18.890,152.927
C06572=1089.554,94.057,437.282,175.383,18.892,152.927
C06573=1089.559,94.306,437.264,175.386,18.893,152.927
C06574=1089.565,94.555,437.246,175.387,18.894,152.926
C06575=1089.570,94.805,437.227,175.389,18.896,152.926
C06576=1089.576,95.054,437.210,175.391,18.897,152.926
C06577=1089.582,95.332,437.190,175.394,18.899,152.926
C06578=1089.589,95.609,437.170,175.396,18.900,152.926
C06579=1089.595,95.885,437.150,175.398,18.902,152.926
C06580=1089.601,96.163,437.130,175.401,18.904,152.926
C06581=1089.607,96.412,437.112,175.403,18.905,152.926
C06582=1089.613,96.662,437.093,175.405,18.907,152.926
C06583=1089.618,96.911,437.075,175.407,18.909,152.926
C06584=1089.624,97.160,437.057,175.409,18.910,152.926
C06585=1089.630,97.409,437.040,175.412,18.911,152.926
C06586=1089.635,97.658,437.021,175.413,18.912,152.925
C06587=1089.641,97.908,437.003,175.416,18.914,152.925
C06588=1089.646,98.157,436.986,175.418,18.915,152.925
C06589=1089.652,98.406,436.966,175.420,18.917,152.925
C06590=1089.658,98.655,436.949,175.422,18.919,152.925
C06591=1089.664,98.905,436.931,175.424,18.920,152.925
C06592=1089.669,99.154,436.913,175.426,18.921,152.925
C06593=1089.675,99.404,436.894,175.429,18.923,152.925
C06594=1089.680,99.653,436.876,175.431,18.924,152.925
C06595=1089.687,99.902,436.858,175.433,18.926,152.925
C06596=1089.692,100.151,436.840,175.435,18.927,152.925
C06597=1089.698,100.401,436.822,175.437,18.928,152.924
C06598=1089.704,100.649,436.803,175.440,18.930,152.924
C06599=1089.709,100.899,436.785,175.441,18.931,152.924
C06600=1089.715,101.148,436.767,175.444,18.933,152.924
C06601=1089.720,101.398,436.748,175.445,18.934,152.924
C06602=1089.726,101.647,436.730,175.448,18.935,152.924
C06603=1089.732,101.896,436.712,175.450,18.937,152.924
C06604=1089.737,102.145,436.694,175.452,18.938,152.924
C06605=1089.743,102.395,436.675,175.454,18.940,152.924
C06606=1089.748,102.644,436.657,175.457,18.941,152.924
C06607=1089.754,102.894,436.639,175.459,18.942,152.923
C06608=1089.759,103.142,436.620,175.461,18.944,152.923
C06609=1089.765,103.392,436.602,175.463,18.945,152.923
C06610=1089.771,103.641,436.583,175.465,18.947,152.923
C06611=1089.776,103.891,436.565,175.468,18.949,152.923
C06612=1089.782,104.139,436.546,175.469,18.950,152.923
C06613=1089.787,104.389,436.528,175.472,18.951,152.923
C06614=1089.793,104.638,436.510,175.474,18.953,152.923
C06615=1089.798,104.888,436.491,175.476,18.954,152.923
C06616=1089.804,105.136,436.473,175.479,18.955,152.923
C06617=1089.810,105.386,436.454,175.480,18.956,152.923
C06618=1089.816,105.635,436.436,175.483,18.958,152.922
C06619=1089.821,105.884,436.417,175.485,18.960,152.922
C06620=1089.827,106.134,436.399,175.487,18.961,152.922
C06621=1089.832,106.383,436.380,175.489,18.962,152.922
C06622=1089.838,106.633,436.361,175.492,18.964,152.922
C06623=1089.843,106.881,436.343,175.493,18.965,152.922
C06624=1089.849,107.131,436.324,175.496,18.967,152.922
C06625=1089.855,107.380,436.306,175.498,18.968,152.922
C06626=1089.860,107.629,436.287,175.500,18.969,152.922
C06627=1089.867,107.878,436.268,175.503,18.971,152.921
C06628=1089.872,108.127,436.250,175.504,18.972,152.921
C06629=1089.877,108.377,436.231,175.507,18.974,152.921
C06630=1089.884,108.626,436.212,175.509,18.975,152.921
C06631=1089.888,108.875,436.194,175.511,18.976,152.921
C06632=1089.895,109.124,436.176,175.514,18.978,152.921
C06633=1089.900,109.373,436.157,175.516,18.979,152.921
C06634=1089.905,109.623,436.138,175.518,18.980,152.921
C06635=1089.912,109.872,436.119,175.520,18.981,152.920
C06636=1089.917,110.121,436.101,175.522,18.982,152.920
C06637=1089.923,110.371,436.083,175.525,18.984,152.920
C06638=1089.929,110.620,436.063,175.527,18.986,152.920
C06639=1089.934,110.869,436.045,175.529,18.987,152.920
C06640=1089.940,111.118,436.026,175.531,18.988,152.920
C06641=1089.946,111.396,436.004,175.534,18.990,152.920
C06642=1089.953,111.673,435.984,175.536,18.991,152.920
C06643=1089.959,111.950,435.964,175.539,18.993,152.919
C06644=1089.965,112.228,435.942,175.541,18.994,152.919
C06645=1089.971,112.477,435.924,175.543,18.996,152.919
C06646=1089.976,112.726,435.905,175.546,18.997,152.919
C06647=1089.982,112.975,435.886,175.548,18.999,152.919
C06648=1089.987,113.224,435.866,175.550,18.999,152.919
C06649=1089.993,113.473,435.848,175.553,19.001,152.919
C06650=1089.999,113.723,435.830,175.555,19.002,152.919
C06651=1090.004,113.972,435.810,175.557,19.003,152.918
C06652=1090.010,114.222,435.791,175.559,19.005,152.918
C06653=1090.016,114.470,435.773,175.562,19.006,152.918
C06654=1090.022,114.720,435.754,175.564,19.007,152.918
C06655=1090.027,114.969,435.734,175.566,19.009,152.918
C06656=1090.032,115.218,435.715,175.569,19.011,152.918
C06657=1090.038,115.467,435.696,175.570,19.012,152.918
C06658=1090.043,115.716,435.677,175.573,19.013,152.918
C06659=1090.049,115.965,435.658,175.575,19.015,152.917
C06660=1090.054,116.215,435.640,175.577,19.016,152.917
C06661=1090.059,116.464,435.621,175.579,19.017,152.917
C06662=1090.065,116.714,435.601,175.582,19.018,152.917
C06663=1090.071,116.963,435.582,175.584,19.019,152.917
C06664=1090.076,117.213,435.563,175.586,19.021,152.917
C06665=1090.081,117.461,435.544,175.589,19.023,152.917
C06666=1090.087,117.711,435.525,175.591,19.024,152.917
C06667=1090.093,117.960,435.506,175.593,19.025,152.916
C06668=1090.098,118.209,435.487,175.596,19.027,152.916
C06669=1090.104,118.458,435.467,175.598,19.028,152.916
C06670=1090.109,118.708,435.448,175.600,19.029,152.916
C06671=1090.115,118.955,435.429,175.603,19.030,152.916
C06672=1090.121,119.205,435.410,175.605,19.032,152.916
C06673=1090.127,119.454,435.391,175.607,19.033,152.916
C06674=1090.132,119.704,435.371,175.609,19.035,152.916
C06675=1090.138,119.953,435.353,175.612,19.036,152.915
C06676=1090.143,120.202,435.333,175.614,19.037,152.915
C06677=1090.149,120.451,435.314,175.616,19.038,152.915
C06678=1090.155,120.701,435.295,175.619,19.040,152.915
C06679=1090.160,120.950,435.276,175.620,19.041,152.915
C06680=1090.165,121.199,435.257,175.623,19.042,152.915
C06681=1090.171,121.448,435.236,175.625,19.044,152.915
C06682=1090.176,121.698,435.217,175.627,19.045,152.914
C06683=1090.182,121.947,435.198,175.630,19.046,152.914
C06684=1090.187,122.196,435.179,175.632,19.048,152.914
C06685=1090.193,122.445,435.160,175.635,19.049,152.914
C06686=1090.198,122.695,435.140,175.637,19.050,152.914
C06687=1090.204,122.943,435.120,175.639,19.051,152.914
C06688=1090.210,123.193,435.101,175.642,19.053,152.913
C06689=1090.215,123.442,435.082,175.644,19.054,152.913
C06690=1090.221,123.691,435.063,175.646,19.055,152.913
C06691=1090.227,123.940,435.043,175.649,19.057,152.913
C06692=1090.233,124.189,435.024,175.651,19.058,152.913
C06693=1090.238,124.439,435.005,175.653,19.059,152.913
C06694=1090.244,124.688,434.985,175.656,19.060,152.912
C06695=1090.250,124.937,434.965,175.658,19.062,152.912
C06696=1090.255,125.186,434.947,175.660,19.062,152.912
C06697=1090.261,125.435,434.927,175.663,19.064,152.912
C06698=1090.267,125.684,434.907,175.665,19.065,152.912
C06699=1090.272,125.934,434.887,175.667,19.066,152.912
C06700=1090.277,126.183,434.868,175.670,19.068,152.912
C06701=1090.283,126.432,434.848,175.672,19.069,152.911
C06702=1090.289,126.681,434.829,175.675,19.070,152.911
C06703=1090.295,126.931,434.810,175.677,19.071,152.911
C06704=1090.301,127.180,434.790,175.679,19.073,152.911
C06705=1090.307,127.457,434.768,175.682,19.074,152.911
C06706=1090.313,127.734,434.746,175.685,19.075,152.911
C06707=1090.320,128.011,434.725,175.687,19.077,152.910
C06708=1090.326,128.288,434.703,175.690,19.078,152.910
C06709=1090.332,128.538,434.684,175.693,19.079,152.910
C06710=1090.337,128.787,434.663,175.694,19.080,152.910
C06711=1090.343,129.036,434.644,175.697,19.082,152.910
C06712=1090.349,129.285,434.624,175.700,19.083,152.909
C06713=1090.354,129.535,434.605,175.702,19.084,152.909
C06714=1090.360,129.783,434.585,175.704,19.085,152.909
C06715=1090.366,130.033,434.566,175.707,19.087,152.909
C06716=1090.371,130.281,434.546,175.709,19.088,152.909
C06717=1090.376,130.531,434.526,175.712,19.089,152.909
C06718=1090.382,130.779,434.506,175.714,19.090,152.908
C06719=1090.388,131.029,434.487,175.716,19.091,152.908
C06720=1090.394,131.278,434.467,175.719,19.092,152.908
C06721=1090.400,131.527,434.448,175.721,19.093,152.908
C06722=1090.405,131.776,434.427,175.723,19.094,152.908
C06723=1090.411,132.026,434.408,175.726,19.096,152.907
C06724=1090.417,132.275,434.388,175.729,19.097,152.907
C06725=1090.422,132.524,434.369,175.730,19.098,152.907
C06726=1090.428,132.773,434.348,175.733,19.099,152.907
C06727=1090.434,133.022,434.328,175.736,19.101,152.907
C06728=1090.439,133.271,434.309,175.738,19.102,152.907
C06729=1090.444,133.520,434.289,175.740,19.103,152.906
C06730=1090.450,133.770,434.269,175.743,19.104,152.906
C06731=1090.455,134.019,434.249,175.745,19.105,152.906
C06732=1090.461,134.268,434.229,175.748,19.107,152.906
C06733=1090.467,134.517,434.210,175.750,19.108,152.906
C06734=1090.472,134.766,434.189,175.752,19.109,152.905
C06735=1090.478,135.015,434.169,175.755,19.110,152.905
C06736=1090.483,135.265,434.149,175.758,19.112,152.905
C06737=1090.489,135.514,434.129,175.760,19.112,152.905
C06738=1090.495,135.763,434.109,175.762,19.114,152.905
C06739=1090.501,136.012,434.089,175.765,19.115,152.904
C06740=1090.506,136.261,434.070,175.767,19.117,152.904
C06741=1090.511,136.510,434.049,175.769,19.117,152.904
C06742=1090.517,136.759,434.029,175.772,19.119,152.904
C06743=1090.523,137.008,434.010,175.775,19.120,152.904
C06744=1090.528,137.258,433.989,175.777,19.121,152.904
C06745=1090.534,137.506,433.969,175.779,19.122,152.903
C06746=1090.540,137.756,433.949,175.782,19.123,152.903
C06747=1090.546,138.005,433.928,175.784,19.124,152.903
C06748=1090.551,138.255,433.909,175.787,19.126,152.903
C06749=1090.557,138.504,433.889,175.789,19.127,152.903
C06750=1090.562,138.753,433.868,175.792,19.128,152.902
C06751=1090.568,139.002,433.848,175.794,19.129,152.902
C06752=1090.574,139.251,433.828,175.797,19.130,152.902
C06753=1090.580,139.499,433.808,175.800,19.131,152.902
C06754=1090.585,139.749,433.788,175.801,19.132,152.902
C06755=1090.591,139.998,433.768,175.804,19.133,152.901
C06756=1090.596,140.247,433.747,175.807,19.135,152.901
C06757=1090.602,140.496,433.727,175.809,19.136,152.901
C06758=1090.607,140.745,433.707,175.811,19.137,152.901
C06759=1090.612,140.994,433.686,175.814,19.138,152.901
C06760=1090.618,141.243,433.666,175.817,19.139,152.900
C06761=1090.624,141.493,433.645,175.819,19.141,152.900
C06762=1090.630,141.742,433.625,175.822,19.142,152.900
C06763=1090.636,141.991,433.605,175.824,19.142,152.900
C06764=1090.640,142.241,433.585,175.826,19.144,152.900
C06765=1090.646,142.489,433.565,175.829,19.145,152.899
C06766=1090.652,142.738,433.544,175.832,19.146,152.899
C06767=1090.657,142.988,433.524,175.833,19.147,152.899
C06768=1090.663,143.236,433.504,175.836,19.148,152.899
C06769=1090.669,143.514,433.480,175.839,19.150,152.899
C06770=1090.676,143.791,433.458,175.841,19.151,152.898
C06771=1090.682,144.068,433.436,175.845,19.153,152.898
C06772=1090.688,144.346,433.413,175.848,19.154,152.898
C06773=1090.694,144.594,433.391,175.850,19.155,152.898
C06774=1090.700,144.843,433.371,175.852,19.156,152.897
C06775=1090.705,145.092,433.351,175.855,19.157,152.897
C06776=1090.710,145.341,433.330,175.858,19.158,152.897
C06777=1090.716,145.590,433.310,175.860,19.159,152.897
C06778=1090.722,145.840,433.289,175.862,19.160,152.897
C06779=1090.727,146.089,433.269,175.865,19.161,152.896
C06780=1090.733,146.338,433.249,175.868,19.163,152.896
C06781=1090.738,146.587,433.228,175.870,19.164,152.896
C06782=1090.744,146.836,433.208,175.873,19.165,152.896
C06783=1090.749,147.085,433.187,175.875,19.165,152.895
C06784=1090.756,147.334,433.166,175.878,19.167,152.895
C06785=1090.761,147.583,433.146,175.880,19.168,152.895
C06786=1090.766,147.832,433.125,175.883,19.169,152.895
C06787=1090.772,148.081,433.105,175.886,19.170,152.894
C06788=1090.779,148.330,433.083,175.888,19.172,152.894
C06789=1090.784,148.579,433.063,175.890,19.172,152.894
C06790=1090.789,148.829,433.042,175.893,19.173,152.894
C06791=1090.794,149.078,433.022,175.896,19.174,152.894
C06792=1090.800,149.327,433.001,175.898,19.176,152.893
C06793=1090.806,149.576,432.980,175.901,19.177,152.893
C06794=1090.812,149.825,432.960,175.903,19.178,152.893
C06795=1090.817,150.074,432.939,175.906,19.179,152.893
C06796=1090.822,150.323,432.919,175.909,19.180,152.892
C06797=1090.828,150.572,432.897,175.911,19.181,152.892
C06798=1090.834,150.821,432.876,175.914,19.182,152.892
C06799=1090.839,151.071,432.856,175.917,19.183,152.892
C06800=1090.844,151.319,432.835,175.918,19.184,152.892
C06801=1090.851,151.569,432.814,175.921,19.186,152.891
C06802=1090.856,151.818,432.794,175.924,19.187,152.891
C06803=1090.862,152.066,432.772,175.927,19.188,152.891
C06804=1090.867,152.315,432.752,175.929,19.189,152.891
C06805=1090.873,152.565,432.731,175.932,19.190,152.890
C06806=1090.879,152.814,432.710,175.934,19.191,152.890
C06807=1090.884,153.063,432.689,175.937,19.192,152.890
C06808=1090.889,153.311,432.668,175.939,19.193,152.890
C06809=1090.895,153.561,432.647,175.942,19.194,152.890
C06810=1090.900,153.810,432.626,175.945,19.195,152.889
C06811=1090.906,154.059,432.605,175.948,19.196,152.889
C06812=1090.912,154.309,432.584,175.949,19.197,152.889
C06813=1090.917,154.557,432.563,175.952,19.198,152.889
C06814=1090.923,154.806,432.542,175.955,19.199,152.888
C06815=1090.929,155.055,432.521,175.958,19.201,152.888
C06816=1090.934,155.304,432.500,175.960,19.202,152.888
C06817=1090.940,155.553,432.479,175.963,19.203,152.888
C06818=1090.946,155.803,432.458,175.965,19.203,152.887
C06819=1090.951,156.051,432.437,175.968,19.204,152.887
C06820=1090.956,156.300,432.416,175.971,19.205,152.887
C06821=1090.963,156.550,432.395,175.973,19.207,152.887
C06822=1090.968,156.799,432.374,175.976,19.208,152.886
C06823=1090.973,157.047,432.353,175.979,19.209,152.886
C06824=1090.979,157.297,432.332,175.981,19.210,152.886
C06825=1090.985,157.546,432.310,175.983,19.211,152.886
C06826=1090.990,157.794,432.289,175.986,19.212,152.885
C06827=1090.996,158.044,432.268,175.989,19.213,152.885
C06828=1091.001,158.293,432.246,175.992,19.214,152.885
C06829=1091.006,158.542,432.226,175.994,19.215,152.885
C06830=1091.012,158.791,432.204,175.997,19.216,152.884
C06831=1091.018,159.040,432.183,176.000,19.217,152.884
C06832=1091.024,159.289,432.162,176.003,19.218,152.884
C06833=1091.030,159.566,432.139,176.005,19.219,152.884
C06834=1091.036,159.843,432.115,176.008,19.220,152.883
C06835=1091.042,160.119,432.091,176.011,19.222,152.883
C06836=1091.049,160.396,432.068,176.014,19.223,152.883
C06837=1091.054,160.646,432.046,176.016,19.224,152.883
C06838=1091.059,160.894,432.025,176.019,19.225,152.882
C06839=1091.066,161.144,432.003,176.022,19.226,152.882
C06840=1091.071,161.392,431.982,176.025,19.227,152.882
C06841=1091.077,161.642,431.961,176.027,19.228,152.882
C06842=1091.082,161.891,431.939,176.030,19.229,152.881
C06843=1091.087,162.139,431.918,176.032,19.230,152.881
C06844=1091.093,162.389,431.897,176.035,19.231,152.881
C06845=1091.098,162.638,431.875,176.038,19.232,152.881
C06846=1091.104,162.886,431.854,176.040,19.233,152.880
C06847=1091.109,163.136,431.832,176.043,19.234,152.880
C06848=1091.115,163.384,431.810,176.046,19.236,152.880
C06849=1091.121,163.634,431.789,176.048,19.237,152.880
C06850=1091.125,163.883,431.768,176.051,19.238,152.879
C06851=1091.131,164.132,431.746,176.054,19.239,152.879
C06852=1091.136,164.381,431.724,176.057,19.240,152.879
C06853=1091.142,164.630,431.703,176.059,19.240,152.879
C06854=1091.148,164.879,431.681,176.061,19.242,152.878
C06855=1091.153,165.128,431.659,176.064,19.243,152.878
C06856=1091.158,165.377,431.639,176.067,19.244,152.878
C06857=1091.164,165.626,431.617,176.070,19.245,152.878
C06858=1091.169,165.875,431.595,176.072,19.246,152.877
C06859=1091.175,166.124,431.573,176.075,19.247,152.877
C06860=1091.180,166.373,431.552,176.078,19.248,152.877
C06861=1091.186,166.622,431.530,176.081,19.249,152.877
C06862=1091.191,166.871,431.508,176.084,19.250,152.876
C06863=1091.197,167.120,431.487,176.086,19.251,152.876
C06864=1091.202,167.369,431.465,176.088,19.252,152.876
C06865=1091.208,167.617,431.444,176.091,19.253,152.876
C06866=1091.213,167.867,431.421,176.094,19.254,152.875
C06867=1091.219,168.115,431.400,176.097,19.255,152.875
C06868=1091.224,168.365,431.378,176.099,19.256,152.875
C06869=1091.230,168.613,431.357,176.102,19.257,152.875
C06870=1091.235,168.863,431.334,176.105,19.258,152.874
C06871=1091.241,169.111,431.313,176.108,19.259,152.874
C06872=1091.246,169.361,431.291,176.110,19.260,152.874
C06873=1091.252,169.610,431.269,176.113,19.262,152.873
C06874=1091.257,169.859,431.247,176.116,19.263,152.873
C06875=1091.263,170.108,431.226,176.119,19.264,152.873
C06876=1091.268,170.356,431.203,176.121,19.265,152.873
C06877=1091.274,170.606,431.181,176.124,19.265,152.872
C06878=1091.279,170.854,431.160,176.126,19.266,152.872
C06879=1091.285,171.104,431.138,176.129,19.267,152.872
C06880=1091.290,171.352,431.116,176.132,19.268,152.872
C06881=1091.296,171.602,431.094,176.135,19.269,152.871
C06882=1091.302,171.851,431.072,176.137,19.270,152.871
C06883=1091.307,172.099,431.050,176.140,19.271,152.871
C06884=1091.313,172.348,431.028,176.143,19.272,152.871
C06885=1091.318,172.597,431.006,176.146,19.273,152.870
C06886=1091.324,172.847,430.984,176.149,19.274,152.870
C06887=1091.329,173.095,430.963,176.151,19.275,152.870
C06888=1091.335,173.344,430.940,176.154,19.276,152.869
C06889=1091.341,173.593,430.918,176.157,19.277,152.869
C06890=1091.346,173.842,430.896,176.160,19.278,152.869
C06891=1091.352,174.091,430.875,176.163,19.279,152.868
C06892=1091.358,174.340,430.852,176.165,19.280,152.868
C06893=1091.363,174.589,430.830,176.168,19.281,152.868
C06894=1091.369,174.838,430.808,176.170,19.282,152.868
C06895=1091.374,175.087,430.785,176.173,19.282,152.867
C06896=1091.380,175.336,430.764,176.176,19.283,152.867
C06897=1091.387,175.612,430.739,176.180,19.285,152.867
C06898=1091.392,175.889,430.715,176.183,19.286,152.866
C06899=1091.399,176.166,430.690,176.185,19.287,152.866
C06900=1091.405,176.442,430.666,176.189,19.288,152.866
C06901=1091.410,176.691,430.644,176.191,19.288,152.865
C06902=1091.416,176.940,430.621,176.194,19.290,152.865
C06903=1091.422,177.189,430.599,176.197,19.291,152.865
C06904=1091.427,177.438,430.577,176.200,19.291,152.865
C06905=1091.433,177.687,430.554,176.202,19.292,152.864
C06906=1091.439,177.936,430.533,176.205,19.293,152.864
C06907=1091.444,178.184,430.510,176.208,19.295,152.864
C06908=1091.449,178.434,430.488,176.211,19.295,152.863
C06909=1091.456,178.682,430.465,176.214,19.296,152.863
C06910=1091.461,178.932,430.443,176.216,19.297,152.863
C06911=1091.467,179.180,430.421,176.219,19.298,152.862
C06912=1091.473,179.429,430.399,176.222,19.299,152.862
C06913=1091.478,179.678,430.376,176.225,19.300,152.862
C06914=1091.484,179.928,430.354,176.228,19.301,152.862
C06915=1091.490,180.176,430.332,176.231,19.302,152.861
C06916=1091.495,180.425,430.310,176.234,19.302,152.861
C06917=1091.501,180.674,430.287,176.236,19.303,152.861
C06918=1091.507,180.923,430.265,176.239,19.305,152.860
C06919=1091.513,181.172,430.242,176.242,19.305,152.860
C06920=1091.518,181.420,430.219,176.245,19.306,152.860
C06921=1091.523,181.670,430.197,176.248,19.307,152.859
C06922=1091.530,181.918,430.175,176.251,19.308,152.859
C06923=1091.535,182.168,430.153,176.253,19.309,152.859
C06924=1091.541,182.417,430.130,176.257,19.310,152.858
C06925=1091.547,182.666,430.107,176.259,19.311,152.858
C06926=1091.552,182.914,430.085,176.262,19.311,152.858
C06927=1091.558,183.163,430.063,176.265,19.312,152.857
C06928=1091.564,183.412,430.040,176.268,19.313,152.857
C06929=1091.569,183.662,430.017,176.271,19.314,152.857
C06930=1091.576,183.910,429.995,176.274,19.315,152.857
C06931=1091.581,184.159,429.972,176.277,19.316,152.856
C06932=1091.587,184.409,429.950,176.279,19.317,152.856
C06933=1091.592,184.657,429.927,176.282,19.317,152.856
C06934=1091.598,184.905,429.905,176.285,19.319,152.855
C06935=1091.604,185.154,429.882,176.288,19.319,152.855
C06936=1091.609,185.404,429.860,176.291,19.320,152.855
C06937=1091.615,185.653,429.837,176.294,19.321,152.854
C06938=1091.621,185.902,429.814,176.297,19.322,152.854
C06939=1091.625,186.150,429.791,176.299,19.323,152.854
C06940=1091.631,186.399,429.768,176.302,19.324,152.853
C06941=1091.636,186.648,429.745,176.305,19.325,152.853
C06942=1091.642,186.897,429.723,176.308,19.326,152.853
C06943=1091.647,187.146,429.700,176.311,19.327,152.853
C06944=1091.653,187.394,429.677,176.313,19.328,152.852
C06945=1091.659,187.643,429.654,176.316,19.329,152.852
C06946=1091.665,187.892,429.631,176.319,19.330,152.852
C06947=1091.670,188.142,429.609,176.322,19.331,152.851
C06948=1091.675,188.391,429.585,176.325,19.331,152.851
C06949=1091.680,188.639,429.563,176.328,19.333,152.851
C06950=1091.686,188.888,429.540,176.330,19.334,152.850
C06951=1091.692,189.137,429.517,176.334,19.335,152.850
C06952=1091.697,189.386,429.494,176.337,19.336,152.850
C06953=1091.703,189.635,429.471,176.340,19.337,152.850
C06954=1091.709,189.884,429.448,176.343,19.338,152.849
C06955=1091.713,190.132,429.425,176.346,19.339,152.849
C06956=1091.719,190.381,429.402,176.348,19.340,152.849
C06957=1091.725,190.630,429.379,176.351,19.340,152.848
C06958=1091.730,190.879,429.356,176.354,19.341,152.848
C06959=1091.736,191.128,429.333,176.357,19.342,152.848
C06960=1091.741,191.377,429.310,176.360,19.343,152.847
C06961=1091.748,191.653,429.284,176.363,19.344,152.847
C06962=1091.754,191.929,429.259,176.366,19.345,152.847
C06963=1091.760,192.206,429.234,176.369,19.346,152.846
C06964=1091.766,192.481,429.208,176.373,19.348,152.846
C06965=1091.771,192.730,429.185,176.376,19.348,152.846
C06966=1091.777,192.979,429.162,176.379,19.349,152.845
C06967=1091.782,193.228,429.138,176.382,19.350,152.845
C06968=1091.788,193.477,429.115,176.385,19.351,152.845
C06969=1091.794,193.726,429.092,176.388,19.352,152.844
C06970=1091.799,193.975,429.069,176.390,19.353,152.844
C06971=1091.804,194.224,429.046,176.393,19.353,152.844
C06972=1091.810,194.473,429.023,176.396,19.354,152.843
C06973=1091.816,194.722,429.000,176.399,19.355,152.843
C06974=1091.822,194.970,428.976,176.402,19.356,152.843
C06975=1091.827,195.219,428.952,176.405,19.357,152.842
C06976=1091.833,195.468,428.930,176.408,19.358,152.842
C06977=1091.838,195.717,428.907,176.410,19.359,152.842
C06978=1091.844,195.966,428.884,176.414,19.360,152.841
C06979=1091.849,196.214,428.859,176.417,19.361,152.841
C06980=1091.855,196.463,428.836,176.420,19.362,152.841
C06981=1091.861,196.712,428.814,176.423,19.362,152.840
C06982=1091.866,196.961,428.789,176.426,19.363,152.840
C06983=1091.872,197.210,428.766,176.429,19.364,152.840
C06984=1091.878,197.458,428.743,176.432,19.365,152.839
C06985=1091.883,197.707,428.720,176.435,19.366,152.839
C06986=1091.889,197.956,428.696,176.437,19.367,152.839
C06987=1091.895,198.206,428.673,176.440,19.368,152.838
C06988=1091.901,198.454,428.650,176.443,19.369,152.838
C06989=1091.906,198.703,428.626,176.447,19.370,152.838
C06990=1091.912,198.952,428.603,176.450,19.370,152.837
C06991=1091.918,199.201,428.580,176.453,19.371,152.837
C06992=1091.923,199.449,428.555,176.456,19.372,152.837
C06993=1091.929,199.698,428.533,176.458,19.373,152.836
C06994=1091.935,199.947,428.509,176.461,19.374,152.836
C06995=1091.940,200.196,428.485,176.464,19.374,152.836
C06996=1091.945,200.445,428.462,176.467,19.376,152.835
C06997=1091.951,200.694,428.438,176.470,19.376,152.835
C06998=1091.957,200.943,428.415,176.473,19.377,152.835
C06999=1091.963,201.191,428.391,176.477,19.378,152.834
C07000=1091.968,201.440,428.368,176.480,19.379,152.834
C07001=1091.974,201.689,428.344,176.483,19.380,152.834
C07002=1091.980,201.938,428.321,176.486,19.381,152.833
C07003=1091.985,202.186,428.297,176.489,19.381,152.833
C07004=1091.991,202.436,428.273,176.491,19.382,152.833
C07005=1091.997,202.684,428.249,176.494,19.383,152.832
C07006=1092.002,202.933,428.226,176.497,19.384,152.832
C07007=1092.008,203.182,428.202,176.501,19.385,152.832
C07008=1092.014,203.430,428.178,176.504,19.386,152.831
C07009=1092.019,203.679,428.155,176.507,19.387,152.831
C07010=1092.025,203.928,428.131,176.510,19.388,152.831
C07011=1092.030,204.177,428.107,176.512,19.389,152.830
C07012=1092.036,204.426,428.083,176.515,19.389,152.830
C07013=1092.042,204.674,428.059,176.518,19.390,152.830
C07014=1092.047,204.924,428.036,176.522,19.392,152.829
C07015=1092.053,205.172,428.012,176.525,19.393,152.829
C07016=1092.058,205.421,427.989,176.528,19.393,152.829
C07017=1092.063,205.670,427.964,176.531,19.394,152.828
C07018=1092.070,205.919,427.940,176.534,19.395,152.828
C07019=1092.075,206.168,427.917,176.537,19.396,152.828
C07020=1092.080,206.416,427.892,176.539,19.397,152.827
C07021=1092.086,206.665,427.869,176.543,19.398,152.827
C07022=1092.091,206.913,427.845,176.546,19.399,152.827
C07023=1092.098,207.163,427.821,176.549,19.400,152.826
C07024=1092.103,207.411,427.797,176.552,19.400,152.826
C07025=1092.126,208.430,427.699,176.613,19.429,152.821
C07026=1092.135,208.808,427.662,176.618,19.433,152.821
C07027=1092.143,209.186,427.625,176.623,19.435,152.821
C07028=1092.152,209.564,427.588,176.627,19.438,152.821
C07029=1092.160,209.941,427.551,176.631,19.440,152.821
C07030=1092.165,210.190,427.527,176.634,19.443,152.821
C07031=1092.171,210.439,427.502,176.637,19.444,152.820
C07032=1092.176,210.688,427.478,176.640,19.446,152.820
C07033=1092.182,210.937,427.453,176.643,19.447,152.820
C07034=1092.188,211.186,427.429,176.646,19.449,152.820
C07035=1092.193,211.434,427.404,176.649,19.451,152.820
C07036=1092.199,211.683,427.379,176.651,19.453,152.820
C07037=1092.204,211.932,427.355,176.655,19.455,152.820
C07038=1092.210,212.180,427.331,176.657,19.456,152.820
C07039=1092.216,212.429,427.307,176.661,19.458,152.819
C07040=1092.222,212.678,427.283,176.663,19.460,152.819
C07041=1092.228,212.926,427.257,176.666,19.462,152.819
C07042=1092.233,213.175,427.233,176.669,19.464,152.819
C07043=1092.238,213.424,427.209,176.672,19.466,152.819
C07044=1092.244,213.673,427.184,176.675,19.467,152.819
C07045=1092.249,213.921,427.159,176.678,19.469,152.819
C07046=1092.255,214.170,427.134,176.681,19.471,152.819
C07047=1092.260,214.419,427.110,176.684,19.473,152.818
C07048=1092.266,214.668,427.085,176.687,19.475,152.818
C07049=1092.272,214.916,427.060,176.689,19.476,152.818
C07050=1092.277,215.165,427.036,176.692,19.478,152.818
C07051=1092.283,215.414,427.011,176.695,19.480,152.818
C07052=1092.289,215.662,426.986,176.698,19.482,152.818
C07053=1092.294,215.912,426.961,176.701,19.484,152.818
C07054=1092.299,216.160,426.937,176.704,19.486,152.818
C07055=1092.305,216.409,426.911,176.707,19.487,152.818
C07056=1092.311,216.658,426.887,176.710,19.489,152.817
C07057=1092.317,216.906,426.862,176.713,19.491,152.817
C07058=1092.322,217.155,426.838,176.716,19.493,152.817
C07059=1092.328,217.403,426.812,176.718,19.495,152.817
C07060=1092.333,217.652,426.787,176.722,19.497,152.817
C07061=1092.339,217.902,426.763,176.724,19.498,152.817
C07062=1092.344,218.150,426.738,176.728,19.501,152.817
C07063=1092.350,218.399,426.713,176.730,19.502,152.817
C07064=1092.356,218.647,426.688,176.734,19.504,152.817
C07065=1092.362,218.896,426.664,176.736,19.506,152.817
C07066=1092.367,219.144,426.638,176.739,19.508,152.816
C07067=1092.373,219.394,426.613,176.742,19.510,152.816
C07068=1092.378,219.642,426.588,176.745,19.512,152.816
C07069=1092.384,219.891,426.564,176.748,19.513,152.816
C07070=1092.389,220.139,426.538,176.751,19.515,152.816
C07071=1092.395,220.388,426.513,176.754,19.517,152.816
C07072=1092.401,220.637,426.488,176.757,19.519,152.816
C07073=1092.407,220.885,426.463,176.760,19.521,152.816
C07074=1092.413,221.134,426.439,176.763,19.523,152.815
C07075=1092.417,221.383,426.413,176.765,19.524,152.815
C07076=1092.424,221.631,426.388,176.769,19.526,152.815
C07077=1092.429,221.880,426.364,176.771,19.528,152.815
C07078=1092.438,222.262,426.325,176.776,19.531,152.815
C07079=1092.446,222.643,426.286,176.781,19.534,152.815
C07080=1092.455,223.025,426.247,176.785,19.536,152.815
C07081=1092.463,223.406,426.208,176.790,19.540,152.814
C07082=1092.470,223.655,426.183,176.792,19.541,152.814
C07083=1092.474,223.904,426.158,176.796,19.543,152.814
C07084=1092.480,224.153,426.133,176.798,19.545,152.814
C07085=1092.485,224.401,426.107,176.802,19.547,152.814
C07086=1092.491,224.650,426.082,176.804,19.548,152.814
C07087=1092.497,224.899,426.056,176.807,19.551,152.814
C07088=1092.502,225.147,426.031,176.811,19.553,152.814
C07089=1092.508,225.396,426.006,176.813,19.554,152.814
C07090=1092.514,225.645,425.980,176.817,19.556,152.813
C07091=1092.519,225.893,425.955,176.819,19.558,152.813
C07092=1092.525,226.142,425.929,176.823,19.560,152.813
C07093=1092.531,226.391,425.905,176.825,19.562,152.813
C07094=1092.536,226.639,425.879,176.828,19.564,152.813
C07095=1092.542,226.888,425.854,176.831,19.565,152.813
C07096=1092.547,227.137,425.828,176.834,19.567,152.813
C07097=1092.553,227.385,425.803,176.837,19.569,152.813
C07098=1092.558,227.634,425.777,176.840,19.571,152.813
C07099=1092.565,227.883,425.752,176.844,19.573,152.812
C07100=1092.570,228.132,425.726,176.846,19.575,152.812
C07101=1092.576,228.380,425.701,176.849,19.577,152.812
C07102=1092.581,228.629,425.675,176.852,19.578,152.812
C07103=1092.587,228.877,425.649,176.855,19.581,152.812
C07104=1092.592,229.125,425.624,176.858,19.582,152.812
C07105=1092.598,229.374,425.598,176.861,19.584,152.812
C07106=1092.604,229.623,425.573,176.864,19.586,152.812
C07107=1092.609,229.872,425.547,176.867,19.588,152.812
C07108=1092.616,230.121,425.521,176.870,19.590,152.812
C07109=1092.620,230.369,425.496,176.873,19.592,152.811
C07110=1092.627,230.618,425.470,176.876,19.594,152.811
C07111=1092.632,230.867,425.444,176.879,19.596,152.811
C07112=1092.638,231.115,425.418,176.882,19.598,152.811
C07113=1092.643,231.363,425.393,176.884,19.600,152.811
C07114=1092.649,231.612,425.367,176.888,19.602,152.811
C07115=1092.654,231.861,425.341,176.891,19.604,152.811
C07116=1092.660,232.110,425.315,176.894,19.605,152.811
C07117=1092.665,232.358,425.290,176.897,19.607,152.811
C07118=1092.671,232.606,425.263,176.900,19.609,152.811
C07119=1092.677,232.855,425.238,176.903,19.611,152.810
C07120=1092.683,233.104,425.212,176.906,19.613,152.810
C07121=1092.688,233.352,425.187,176.909,19.615,152.810
C07122=1092.693,233.601,425.161,176.912,19.617,152.810
C07123=1092.699,233.850,425.134,176.915,19.618,152.810
C07124=1092.705,234.099,425.108,176.918,19.621,152.810
C07125=1092.711,234.347,425.083,176.920,19.623,152.810
C07126=1092.716,234.596,425.056,176.924,19.625,152.810
C07127=1092.721,234.844,425.031,176.927,19.627,152.810
C07128=1092.727,235.093,425.005,176.929,19.628,152.810
C07129=1092.732,235.342,424.979,176.933,19.631,152.810
C07130=1092.741,235.715,424.939,176.937,19.633,152.809
C07131=1092.750,236.088,424.901,176.942,19.637,152.809
C07132=1092.758,236.461,424.861,176.946,19.639,152.809
C07133=1092.766,236.833,424.822,176.951,19.643,152.809
C07134=1092.772,237.082,424.796,176.954,19.644,152.809
C07135=1092.777,237.331,424.770,176.957,19.646,152.809
C07136=1092.783,237.579,424.743,176.959,19.648,152.809
C07137=1092.788,237.828,424.717,176.963,19.650,152.809
C07138=1092.795,238.076,424.691,176.966,19.652,152.808
C07139=1092.800,238.325,424.665,176.969,19.654,152.808
C07140=1092.806,238.574,424.639,176.972,19.656,152.808
C07141=1092.812,238.823,424.613,176.974,19.658,152.808
C07142=1092.817,239.070,424.587,176.978,19.660,152.808
C07143=1092.822,239.319,424.561,176.981,19.662,152.808
C07144=1092.828,239.567,424.534,176.984,19.664,152.808
C07145=1092.834,239.816,424.507,176.987,19.666,152.808
C07146=1092.839,240.065,424.481,176.990,19.668,152.808
C07147=1092.845,240.313,424.455,176.993,19.669,152.808
C07148=1092.850,240.562,424.429,176.996,19.671,152.808
C07149=1092.856,240.811,424.402,177.000,19.674,152.807
C07150=1092.862,241.059,424.376,177.002,19.675,152.807
C07151=1092.867,241.308,424.350,177.005,19.678,152.807
C07152=1092.873,241.556,424.323,177.008,19.679,152.807
C07153=1092.879,241.805,424.296,177.011,19.681,152.807
C07154=1092.884,242.054,424.270,177.014,19.684,152.807
C07155=1092.890,242.302,424.244,177.017,19.685,152.807
C07156=1092.896,242.550,424.217,177.020,19.687,152.807
C07157=1092.901,242.799,424.191,177.024,19.689,152.807
C07158=1092.907,243.048,424.165,177.026,19.691,152.807
C07159=1092.913,243.296,424.138,177.030,19.693,152.807
C07160=1092.919,243.544,424.111,177.033,19.696,152.807
C07161=1092.924,243.794,424.085,177.035,19.697,152.806
C07162=1092.929,244.042,424.058,177.039,19.699,152.806
C07163=1092.935,244.290,424.031,177.042,19.701,152.806
C07164=1092.941,244.539,424.005,177.044,19.703,152.806
C07165=1092.947,244.787,423.978,177.048,19.706,152.806
C07166=1092.952,245.036,423.952,177.051,19.708,152.806
C07167=1092.957,245.285,423.925,177.053,19.709,152.806
C07168=1092.963,245.533,423.898,177.057,19.711,152.806
C07169=1092.969,245.781,423.872,177.060,19.713,152.806
C07170=1092.974,246.030,423.845,177.062,19.716,152.806
C07171=1092.980,246.278,423.818,177.066,19.718,152.806
C07172=1092.985,246.527,423.791,177.069,19.720,152.806
C07173=1092.991,246.775,423.764,177.072,19.721,152.806
C07174=1092.997,247.024,423.738,177.075,19.723,152.805
C07175=1093.002,247.272,423.711,177.078,19.726,152.805
C07176=1093.008,247.521,423.684,177.081,19.728,152.805
C07177=1093.014,247.770,423.657,177.084,19.730,152.805
C07178=1093.019,248.018,423.630,177.087,19.732,152.805
C07179=1093.025,248.267,423.603,177.090,19.734,152.805
C07180=1093.031,248.515,423.576,177.093,19.736,152.805
C07181=1093.036,248.764,423.549,177.096,19.738,152.805
C07182=1093.044,249.130,423.510,177.100,19.741,152.805
C07183=1093.052,249.496,423.470,177.105,19.744,152.805
C07184=1093.060,249.862,423.431,177.110,19.747,152.805
C07185=1093.068,250.228,423.390,177.114,19.751,152.805
C07186=1093.074,250.476,423.363,177.117,19.752,152.805
C07187=1093.079,250.725,423.336,177.120,19.754,152.804
C07188=1093.085,250.973,423.309,177.123,19.757,152.804
C07189=1093.090,251.222,423.283,177.126,19.758,152.804
C07190=1093.095,251.470,423.256,177.129,19.761,152.804
C07191=1093.101,251.719,423.229,177.132,19.763,152.804
C07192=1093.107,251.968,423.201,177.136,19.765,152.804
C07193=1093.113,252.216,423.174,177.138,19.767,152.804
C07194=1093.118,252.465,423.147,177.142,19.769,152.804
C07195=1093.124,252.713,423.120,177.145,19.771,152.804
C07196=1093.129,252.961,423.092,177.147,19.773,152.804
C07197=1093.135,253.209,423.065,177.151,19.775,152.804
C07198=1093.141,253.459,423.038,177.154,19.778,152.804
C07199=1093.147,253.706,423.010,177.157,19.780,152.804
C07200=1093.152,253.955,422.983,177.160,19.781,152.804
C07201=1093.157,254.203,422.957,177.163,19.783,152.804
C07202=1093.163,254.452,422.929,177.166,19.786,152.804
C07203=1093.169,254.701,422.902,177.169,19.788,152.803
C07204=1093.174,254.949,422.874,177.172,19.790,152.803
C07205=1093.180,255.197,422.846,177.175,19.792,152.803
C07206=1093.185,255.446,422.820,177.179,19.794,152.803
C07207=1093.191,255.695,422.792,177.181,19.796,152.803
C07208=1093.197,255.943,422.765,177.184,19.798,152.803
C07209=1093.202,256.191,422.738,177.188,19.801,152.803
C07210=1093.208,256.439,422.710,177.191,19.803,152.803
C07211=1093.214,256.689,422.683,177.193,19.804,152.803
C07212=1093.219,256.937,422.655,177.197,19.806,152.803
C07213=1093.225,257.185,422.628,177.200,19.809,152.803
C07214=1093.230,257.433,422.600,177.203,19.811,152.803
C07215=1093.237,257.682,422.573,177.206,19.813,152.803
C07216=1093.242,257.930,422.545,177.209,19.815,152.803
C07217=1093.247,258.179,422.518,177.212,19.817,152.803
C07218=1093.254,258.427,422.490,177.216,19.820,152.802
C07219=1093.259,258.676,422.463,177.218,19.821,152.802
C07220=1093.265,258.924,422.435,177.221,19.824,152.802
C07221=1093.271,259.172,422.407,177.225,19.826,152.802
C07222=1093.276,259.421,422.380,177.228,19.828,152.802
C07223=1093.282,259.669,422.353,177.231,19.829,152.802
C07224=1093.288,259.918,422.324,177.234,19.832,152.802
C07225=1093.293,260.166,422.297,177.237,19.834,152.802
C07226=1093.299,260.414,422.270,177.240,19.836,152.802
C07227=1093.305,260.663,422.241,177.243,19.838,152.802
C07228=1093.310,260.911,422.214,177.246,19.840,152.802
C07229=1093.317,261.160,422.186,177.249,19.843,152.802
C07230=1093.322,261.408,422.158,177.253,19.845,152.802
C07231=1093.327,261.657,422.131,177.255,19.847,152.802
C07232=1093.334,261.905,422.103,177.258,19.849,152.802
C07233=1093.339,262.153,422.075,177.262,19.851,152.802
C07234=1093.347,262.517,422.034,177.266,19.854,152.801
C07235=1093.356,262.879,421.994,177.271,19.857,152.801
C07236=1093.364,263.243,421.953,177.276,19.860,152.801
C07237=1093.372,263.606,421.913,177.280,19.863,152.801
C07238=1093.379,263.855,421.885,177.283,19.865,152.801
C07239=1093.384,264.103,421.857,177.287,19.868,152.801
C07240=1093.390,264.351,421.829,177.289,19.869,152.801
C07241=1093.396,264.599,421.801,177.292,19.872,152.801
C07242=1093.401,264.848,421.773,177.296,19.874,152.801
C07243=1093.407,265.096,421.744,177.299,19.876,152.801
C07244=1093.413,265.345,421.718,177.302,19.879,152.801
C07245=1093.419,265.593,421.689,177.304,19.881,152.801
C07246=1093.424,265.841,421.661,177.308,19.883,152.801
C07247=1093.429,266.089,421.633,177.311,19.885,152.801
C07248=1093.435,266.338,421.605,177.314,19.887,152.801
C07249=1093.441,266.586,421.577,177.318,19.889,152.801
C07250=1093.447,266.835,421.549,177.320,19.892,152.801
C07251=1093.452,267.083,421.521,177.323,19.894,152.801
C07252=1093.458,267.332,421.492,177.326,19.896,152.801
C07253=1093.464,267.579,421.464,177.330,19.898,152.801
C07254=1093.469,267.828,421.435,177.333,19.901,152.801
C07255=1093.475,268.076,421.408,177.335,19.902,152.800
C07256=1093.481,268.325,421.379,177.339,19.905,152.800
C07257=1093.486,268.573,421.351,177.342,19.907,152.800
C07258=1093.492,268.822,421.323,177.345,19.909,152.800
C07259=1093.497,269.070,421.295,177.348,19.912,152.800
C07260=1093.503,269.318,421.267,177.352,19.914,152.800
C07261=1093.509,269.566,421.238,177.354,19.916,152.800
C07262=1093.514,269.815,421.209,177.357,19.918,152.800
C07263=1093.520,270.063,421.181,177.360,19.921,152.800
C07264=1093.525,270.312,421.153,177.364,19.923,152.800
C07265=1093.531,270.560,421.125,177.367,19.925,152.800
C07266=1093.537,270.808,421.096,177.370,19.927,152.800
C07267=1093.542,271.056,421.068,177.373,19.929,152.800
C07268=1093.548,271.305,421.039,177.376,19.932,152.800
C07269=1093.554,271.553,421.012,177.379,19.934,152.800
C07270=1093.559,271.801,420.982,177.382,19.936,152.800
C07271=1093.565,272.050,420.954,177.386,19.939,152.800
C07272=1093.570,272.298,420.926,177.389,19.941,152.800
C07273=1093.577,272.546,420.897,177.391,19.943,152.800
C07274=1093.582,272.794,420.869,177.395,19.945,152.800
C07275=1093.587,273.043,420.840,177.398,19.948,152.800
C07276=1093.593,273.291,420.811,177.401,19.950,152.800
C07277=1093.599,273.539,420.783,177.404,19.952,152.800
C07278=1093.605,273.788,420.754,177.407,19.955,152.800
C07279=1093.610,274.036,420.726,177.411,19.957,152.800
C07280=1093.616,274.285,420.697,177.413,19.959,152.800
C07281=1093.621,274.532,420.668,177.416,19.961,152.800
C07282=1093.627,274.781,420.640,177.420,19.964,152.800
C07283=1093.633,275.029,420.610,177.423,19.966,152.800
C07284=1093.638,275.277,420.582,177.426,19.968,152.800
C07285=1093.644,275.525,420.553,177.429,19.971,152.800
C07286=1093.653,275.919,420.508,177.434,19.975,152.800
C07287=1093.662,276.314,420.462,177.439,19.978,152.800
C07288=1093.671,276.707,420.416,177.444,19.982,152.800
